(* PLC project Ackersteuerung, ForgeIEC ForgeIEC 0.1.0, author Jörg Bernau *)
(* stored: creationDateTime 2026-08-31T00:10:50 *)
(* # Ackersteuerung — Bewässerungssteuerung des SoLaWi-Ackers „Ackervielfalt"

> Automatisierte, bedarfsgerechte Bewässerung des Gemeinschaftsackers der SoLaWi Ackervielfalt
> (Kooperation mit **SALZ Automation** ). Ziel: präzises, wassersparendes Bewässern statt Handgießen.
> Ref: https://www.solawi-ackervielfalt.de/kooperation-salz-automation/
>
> Repository: https://github.com/Beerlesklopfer/Ackervielfalt — SPS-Projekt `Ackersteuerung.forge`,
> HMI-Projekt `Ackersteuerung.hearth`. **Stand 2026-09-29.**

---

## 0. Harte Randbedingungen

1. **Höchstens `Betrieb.uMaxVentile` Ventile gleichzeitig offen** (Startwert 24) — erzwungen
   durch `FB_TERMINAL_OUT` über alle Betriebsarten.
2. **Kein angewähltes Beet wird ausgelassen** — die Laufzeit zählt erst, wenn das Ventil wirklich
   offen ist; ein Beet wartet höchstens, es wird nie übersprungen.
3. **Genau eine Betriebsart** — `Betrieb.uModeActive` trägt je Betriebsart ein Bit; 0 = AUS
   (alle Ventile zu).
4. **Anwahl per HMI oder Taster** am Beet, gleichberechtigt (Dual-Namespace `Anvil.*` Hardware /
   `Bellows.*` HMI).

## 1. Anlage und Bus

Sechs Feldboxen (Amsamotion Modbus-TCP) und ein Weidmüller-UR20-Koppler, zwei Segmente an `end0`:

| Gerät | Typ | IP | Segment | Index |
|---|---|---|---|---|
| Pfirsich | ETH-MODBUS-IO8R-A | .26 | MODBUS-SUED | 0–3 |
| Stachelbeere | ETH-MODBUS-IO8R-A | .28 | MODBUS-SUED | 4–7 |
| Maulbeere | ETH-MODBUS-IO8R-A | .29 | MODBUS-SUED | 8–11 |
| Felsenbirne | ETH-MODBUS-IO8R-A | .27 | MODBUS-SUED | 12–15 |
| Maibeere | ETH-MODBUS-IO8R-A | .25 | MODBUS_NORD | 16–19 |
| Johannisbeere | ETH-MODBUS-IO8R-A | .24 | MODBUS_NORD | 20–23 |
| Schaltschrank | Weidmüller UR20-FBC-MOD-TCP (8 DI / 8 DO) | .229 | MODBUS_NORD | — |

Netz 192.168.24.x. **Alle Felder je Ventil laufen 0..23**, Index `i = z*4 + v` (Zone z in der
Reihenfolge der Tabelle, v = Taster/Ventil − 1). Die Zuordnung legt `FB_TERMINAL_OUT` fest.

## 2. Ein- und Ausgänge je Feldbox

IO8R-A (alle sechs Feldboxen): `xT_1..4` Beet-Taster · `xT_5..8` frei · `xV_1..4` Ventile ·
`xLed_5..8` Status-LEDs der Ventile 1..4 · `wAI_Voltage_1..3`, `wAI_Current_1..3`
Analogeingänge · `wAO_1..2` Analogausgänge.

## 3. Betriebsarten (`Betrieb.uModeActive`)

`PLC_PRG` ruft jeden Modus-Baustein in jedem Zyklus; sein `xEnable` entscheidet, ob er arbeitet.
Ein abgeschalteter Baustein friert ein. Dasselbe Bit setzt jeder Baustein als `bModeBit` je Ventil
in `Betrieb.astValveStatus[i].bMode`.

| Bit | Betriebsart | Baustein | Verhalten |
|---|---|---|---|
| 0 | AUS | — | nichts vorgewählt, alle Ventile und LEDs aus |
| 1 | Manuell | `fbManual` : `FB_MANUAL` | Taster oder HMI schalten das Ventil um |
| 2 | One-Shot | `fbOneShot` : `FB_SCHEDULE` | angewählte Beete laufen nach Start einmal ihre Dauer |
| 4 | wiederkehrend | `fbRecurring` : `FB_SCHEDULE` | wie One-Shot; Startzeit und Wochentage noch nicht ausgewertet (§10) |
| 8 | Auto | `fbAuto` : `FB_WEEKLY_TIMER` | Platzhalter, Bedarf nach Kc/ET0 zurückgestellt; öffnet kein Ventil |

### Lauf in One-Shot und wiederkehrend (`FB_SCHEDULE`)

- **Anwahl:** je Beet ein `JK_FF`; Feldtaster `Anvil.<Zone>.xT_v` und HMI-Puls
  `Schrittkette.axSelToggle[i]` schalten gleichberechtigt um. Q ist `Betrieb.aValveJobs[i].xSelected`.
  Nicht persistent.
- **Befehle** (je eine steigende Flanke): `Schrittkette.xStart`, `xStop`, `xPause`, `xAcknowledge`.
- **Zustand** `Schrittkette.uRunState`: 0 Idle · 1 Running · 2 Paused · 3 Done.
- **Timer:** je Beet ein `TONR` (pausierbar). Er zählt nur, solange Running und das Ventil wirklich
  offen ist; Pause und Warten auf Freigabe halten ihn an.
- **Restzeit:** `Betrieb.astValveStatus[i].remainingLiquidation` = PT − ET, nicht persistent; die HMI liest sie dort direkt.

## 4. Ausgabe und Anzeige (`FB_TERMINAL_OUT`)

`FB_TERMINAL_OUT` ist der eine Setter: Vorwahl der aktiven Betriebsart, Arbitrierung, 48 Klemmen.

- Laufende Freigaben **halten**, solange vorgewählt; neue nur bei freiem Platz, in
  Index-Reihenfolge, ohne Verdrängung.
- Fällt ein offenes Ventil, ist die Vorwahl **verbraucht** (das Bit der Betriebsart fällt).
- Ventile `xV_1..4` folgen allein der Freigabe (`astValveStatus[i].isOpen`).
- LEDs `xLed_5..8`: Dauerlicht = offen; vorgewählt und wartend = Blinken im Takt
  `Betrieb.rBlinkHz` (Startwert 0.1 Hz, begrenzt auf 0.01..10 Hz).

## 5. Persistente Einstellungen

Persistent heißt: der Wert übersteht Neustart und Programm-Download. Alle sind von der HMI
schreibbar.

| Variable | Label | Startwert | Bedeutung |
|---|---|---|---|
| `Betrieb.uModeActive` | Aktive Betriebsart | 0 | Bit der Betriebsart (§3) |
| `Betrieb.uMaxVentile` | Max. offene Ventile | 24 | Höchstzahl gleichzeitig offener Ventile |
| `Betrieb.rBlinkHz` | Blinkfrequenz wartende Ventile [Hz] | 0.1 | Blinktakt wartender Ventile |
| `Betrieb.aValveJobs` | Ventil-Jobs | Dauer 1 min | je Beet `ST_BedCfg`: Anwahl, Startzeit, Dauer |
| `Betrieb.bWeekMask` | Wochentage wiederkehrend | 0 | Bit 0 = Montag … Bit 6 = Sonntag |

**Achtung:** Gespeichert wird je Variable mit einer Typkennung. Ändert sich der Typ (ein Feld mehr
in `ST_BedCfg`, andere Feldgrenzen), verwirft der nächste Download die gespeicherten Werte dieser
Variable einmal.

## 6. HMI-Gruppen

- `Betrieb`: Einstellungen (§5) und `astValveStatus[0..23]` (`ST_ValveStatus`: bMode,
  isPreselected, isOpen, liquidationPeriod, remainingLiquidation).
- `Schrittkette`: `axSelToggle[0..23]`, die vier Befehle, `uRunState`.
- `Diag`: Geräteüberwachung (§7).
- `HmiCmd`: leer.

## 7. Geräteüberwachung

`BusMonitor` (taskDiag) liest je Gerät `Anvil.<Gerät>.Status.xOnline`, `FB_BUS_MONITOR` führt je
Gerät einen `FB_DEVICE_MONITOR` (0 Unbekannt → 1 Online → 2 Gestört → 3 Offline, entprellt) und
schreibt nach `Bellows.Diag`: `auDevState[0..6]`, `asDevStatus`, `sSummary`, `xAllOk`,
`iFaultCount`. Index 0 Pfirsich … 5 Johannisbeere, 6 Schaltschrank — handgepflegt.

## 8. Tasks

| Task | Takt | Priorität | Programm |
|---|---|---|---|
| task0 | 20 ms | 0 | `PLC_PRG` |
| taskDiag | 200 ms | 10 | `BusMonitor` |

## 9. Bausteine und Typen

Programme: `PLC_PRG`, `BusMonitor`. Funktionsbausteine: `FB_MANUAL`, `FB_SCHEDULE`,
`FB_TERMINAL_OUT`, `FB_BLINK`, `FB_WEEKLY_TIMER`, `FB_DEVICE_MONITOR`, `FB_BUS_MONITOR`.
Funktion: `FC_GetKcValue`. Aus der Standardbibliothek u. a. `JK_FF`, `TONR`, `R_TRIG`, `TON`.
Gruppen: sieben Geräte (Pfirsich … Schaltschrank) und die HMI-Gruppen `Betrieb`, `Schrittkette`,
`Diag`, `HmiCmd`.
Typen: `ST_BedCfg` (xSelected, uStartHour, uStartMin, tDuration), `ST_ValveStatus`,
`ST_KcCurve`.

## 10. Offene Punkte (2026-09-29)

- **Wochenschaltuhr:** Betriebsart wiederkehrend wertet `uStartHour`, `uStartMin` und
  `bWeekMask` noch nicht aus — sie läuft wie One-Shot auf Start. Die Dialoge zeigen bis dahin nur
  Anwahl und Dauer.
- `HmiCmd` ist leer.
- Schaltschrank: Ein- und Ausgänge ungenutzt; die Bindungen stehen in der alten Steckplatz-Zählung
  (Stand 2026-09-11, nicht neu geprüft).
- Analogausgänge `wAO_1..2`: die Bindung nennt Register 0/1, die Gerätebeschreibung 6/7
  (Stand 2026-09-11, nicht neu geprüft).
- Betriebsart Auto (Kc/ET0) wartet auf Wetter- und Bodensensorik. *)

TYPE ST_KcCurve : STRUCT
  days_initial : INT;
  days_dev : INT;
  days_mid : INT;
  days_late : INT;
  kc_initial : REAL;
  kc_mid : REAL;
  kc_end : REAL;
END_STRUCT;
END_TYPE

(* Ein Beet (ein Ventil) fuer One-Shot und wiederkehrend: Anwahl, Startzeit in Ortszeit und Bewaesserungsdauer (Vorgabe 1 min). Element der persistenten Job-Liste Betrieb.aValveJobs[0..23], Index z*4+v. xSelected schreibt die SPS (FB_SCHEDULE), Startzeit und Dauer die HMI. Die laufende Restzeit steht NICHT hier, sondern im nicht persistenten Betrieb.astValveStatus[i].remainingLiquidation — sie aendert sich jeden Zyklus, und in einem persistenten Satz schrieb sie im Lauf alle 5 s die Persistenzdatei (29.09.2026). *)
TYPE ST_BedCfg : STRUCT
  xSelected : BOOL := FALSE;  (* Wird dieses Beet bei der bewässerung berücksichtigt? *)
  uStartHour : BYTE;  (* Startzeit Stunde (Ortszeit) *)
  uStartMin : BYTE;  (* Startzeit Minute *)
  tDuration : TIME := T#1m;  (* Bewaesserungsdauer dieses Ventils, Vorgabe 1 min *)
END_STRUCT;
END_TYPE

(* Status je Ventil (Betrieb.astValveStatus, Index z*4+v). bMode: je Betriebsart ein Bit (1 Manuell, 2 One-Shot, 4 wiederkehrend, 8 Auto), von jedem Modus-Baustein in seiner Schleife gesetzt. isPreselected: vorgewaehlt in der AKTIVEN Betriebsart, (bMode AND GVL.Betrieb.uModeActive) <> 0 — schreibt FB_TERMINAL_OUT. isOpen: wirklich offen = Freigabe der Arbitrierung in FB_TERMINAL_OUT (nie mehr als uMaxVentile, laufende halten, nachruecken in Index-Reihenfolge); haelt ueber die Zyklen. liquidationPeriod: eingestellte Laufdauer, vom Modus (Manuell T#0s = unbegrenzt). remainingLiquidation: Restlauf = liquidationPeriod − ET des Modus-Timers, vom Modus berechnet. *)
TYPE ST_ValveStatus : STRUCT
  bMode : BYTE := 0;
  isPreselected : BOOL := FALSE;
  isOpen : BOOL := FALSE;
  liquidationPeriod : TIME := T#0s;
  remainingLiquidation : TIME := T#0s;
END_STRUCT;
END_TYPE

(* HMI-Gruppe Betrieb: Betriebsartwahl xManuell, xOneShot, xWiederkehrend, xAuto (genau eine gesetzt, sonst Aus), die bestaetigte Betriebsart uModeActive (0 Aus, 1 Manuell, 2 One-Shot, 3 wiederkehrend, 4 Auto) und die Einstellwerte uMaxVentile und rBlinkHz. Wahl und Einstellwerte sind persistent. *)
PROGRAM Betrieb
  VAR_GLOBAL
    uModeActive AT %MB0 : USINT := 0;  (* Aktive Betriebsart, je Betriebsart ein Bit: 0 = AUS, 1 = Manuell, 2 = One-Shot, 4 = wiederkehrend, 8 = Auto. Die EINE Quelle: PLC_PRG gibt damit die Modus-Bausteine frei (xEnable) und reicht dasselbe Bit als bModeBit weiter; FB_TERMINAL_OUT liest damit die Vorwahl aus astValveStatus[i].bMode. Von der HMI gesetzt, persistent. *)
    uMaxVentile AT %MB2 : USINT := 24;  (* Hoechstzahl gleichzeitig offener Ventile (Wasserdruck, Pumpenleistung). FB_TERMINAL_OUT begrenzt auf diese Zahl; weitere Anforderungen warten in Index-Reihenfolge und ruecken nach, sobald ein Platz frei wird. Startwert 24. Von der HMI gesetzt, persistent. *)
    rBlinkHz AT %MD7 : REAL := 0.1;  (* Blinkfrequenz der Status-LEDs wartender Ventile in den Betriebsarten Manuell, One-Shot und wiederkehrend, in Hz: angefordert, aber vom Arbiter noch nicht freigegeben. PLC_PRG begrenzt auf 0.01..10 Hz, ein Wert unter 0.01 gilt als 0.1. Startwert 0.1 Hz = 5 s an / 5 s aus. Von der HMI gesetzt, persistent. *)
  END_VAR

            
          
END_PROGRAM

(* # FB_BLINK — Blink-/Flash-Generator (Programm-Anzeige) Asymmetrisches Blinksignal aus zwei TON: kurzer Flash (`tBlFlash`) + längere Pause (`tBlPause`); `xBlQ` ist Phasen-Bit + Ausgang. `xBlEnable=FALSE` hält `xBlQ` dauerhaft FALSE (Handbetrieb blinkt nicht). In PLC_PRG mit `T#1S`/`T#29S` ( **Periode 30 s** ) für die Programm-Anzeige `xV_6..8` parametriert. Review-Hinweis: bei Enable startet die Pause zuerst (erster Flash nach `tBlPause`); `PT=0` ungeguardet. *)
FUNCTION_BLOCK FB_BLINK
  VAR
    tonBlOn : TON;  (* Timer für Flash-Dauer (tBlFlash) *)
    tonBlOff : TON;  (* Timer für Pausen-Dauer (tBlPause) *)
    xWasEnabled : BOOL;  (* Flankenspeicher xBlEnable: bei steigender Flanke startet die Anzeige mit einem Flash (sofortige Rueckmeldung) *)
  END_VAR
  VAR_INPUT
    xBlEnable : BOOL;  (* Blinken aktiv; FALSE = xBlQ dauerhaft FALSE (z. B. Handbetrieb) *)
    tBlFlash : TIME := T#1S;  (* Kurzer Flash (Ein-Dauer); relais-schonend: 1 s Flash bei 10 s Periode (1 s ein / 9 s aus) *)
    tBlPause : TIME := T#9S;  (* Laengere Pause (Aus-Dauer); relais-schonend: 9 s Pause bei 10 s Periode (1 s ein / 9 s aus) *)
  END_VAR
  VAR_OUTPUT
    xBlQ : BOOL;  (* Blink-Ausgang: kurzer Flash, längere Pause; FALSE bei NOT xBlEnable *)
  END_VAR

            (* Disable: Ausgang sofort aus, Flankenspeicher zuruecksetzen. *)
IF NOT xBlEnable THEN
    xBlQ := FALSE;
    xWasEnabled := FALSE;
ELSIF NOT xWasEnabled THEN
    (* Steigende Flanke von Enable: mit einem Flash STARTEN -> sofortige
       Rueckmeldung, kein Warten auf die erste Pause. Relais-schonend 1s/9s. *)
    xBlQ := TRUE;
    xWasEnabled := TRUE;
END_IF;

(* Zwei TON bilden den asymmetrischen Oszillator:
     - waehrend Flash (xBlQ=TRUE)  laeuft tonBlOn  (PT=tBlFlash)
     - waehrend Pause (xBlQ=FALSE) laeuft tonBlOff (PT=tBlPause) *)
tonBlOn (IN := xBlEnable AND xBlQ,     PT := tBlFlash);
tonBlOff(IN := xBlEnable AND NOT xBlQ, PT := tBlPause);

IF xBlEnable THEN
    IF xBlQ AND tonBlOn.Q THEN
        xBlQ := FALSE;          (* Flash zu Ende -> Pause beginnt *)
    ELSIF (NOT xBlQ) AND tonBlOff.Q THEN
        xBlQ := TRUE;           (* Pause zu Ende -> Flash beginnt *)
    END_IF;
END_IF;
          
END_FUNCTION_BLOCK

(* Feldbox Felsenbirne (Amsamotion ETH-MODBUS-IO8R-A, 192.168.24.27, Segment MODBUS-SUED), Ventile 13-16 der Job-Liste. xT_1..4 Beet-Taster, xT_5..8 frei; xV_1..4 Ventile (= Arbiter-Freigabe); xV_5..8 Status-LEDs der Ventile 1..4; wAI_Voltage_1..3 und wAI_Current_1..3 Analogeingaenge; wAO_1..2 Analogausgaenge. Anvil.* ist die Hardware-Sicht, Bellows.* die HMI-Sicht derselben Variablen. *)
PROGRAM Felsenbirne
  VAR_GLOBAL
    xT_1 AT %IX5.0 : BOOL;  (* Digital input channel 1 (24V DC, opto-isolated) *)
    xT_2 AT %IX5.1 : BOOL;  (* Digital input channel 2 (24V DC, opto-isolated) *)
    xT_3 AT %IX5.2 : BOOL;  (* Digital input channel 3 (24V DC, opto-isolated) *)
    xT_4 AT %IX5.3 : BOOL;  (* Digital input channel 4 (24V DC, opto-isolated) *)
    xT_5 AT %IX5.4 : BOOL;  (* Digital input channel 5 (24V DC, opto-isolated) *)
    xT_6 AT %IX5.5 : BOOL;  (* Digital input channel 6 (24V DC, opto-isolated) *)
    xT_7 AT %IX5.6 : BOOL;  (* Digital input channel 7 (24V DC, opto-isolated) *)
    xT_8 AT %IX5.7 : BOOL;  (* Digital input channel 8 (24V DC, opto-isolated) *)
    xV_1 AT %QX5.0 : BOOL;  (* Relay output channel 1 (max 2A) *)
    xV_2 AT %QX5.1 : BOOL;  (* Relay output channel 2 (max 2A) *)
    xV_3 AT %QX5.2 : BOOL;  (* Relay output channel 3 (max 2A) *)
    xV_4 AT %QX5.3 : BOOL;  (* Relay output channel 4 (max 2A) *)
    xLed_5 AT %QX5.4 : BOOL;  (* Relay output channel 5 (max 2A) *)
    xLed_6 AT %QX5.5 : BOOL;  (* Relay output channel 6 (max 2A) *)
    xLed_7 AT %QX5.6 : BOOL;  (* Relay output channel 7 (max 2A) *)
    xLed_8 AT %QX5.7 : BOOL;  (* Relay output channel 8 (max 2A) *)
    wAO_1 AT %QW8 : UINT;  (* Analog output channel 1 (0-10V / 0-20mA, 12-bit) *)
    wAO_2 AT %QW9 : UINT;  (* Analog output channel 2 (0-10V / 0-20mA, 12-bit) *)
    wAI_Voltage_1 AT %IW24 : UINT;  (* Analog input channel 1 (0-10V, 12-bit) *)
    wAI_Voltage_2 AT %IW25 : UINT;  (* Analog input channel 2 (0-10V, 12-bit) *)
    wAI_Voltage_3 AT %IW26 : UINT;  (* Analog input channel 3 (0-10V, 12-bit) *)
    wAI_Current_1 AT %IW27 : UINT;  (* Analog input channel 4 (0-20mA, 12-bit) *)
    wAI_Current_2 AT %IW28 : UINT;  (* Analog input channel 5 (0-20mA, 12-bit) *)
    wAI_Current_3 AT %IW29 : UINT;  (* Analog input channel 6 (0-20mA, 12-bit) *)
  END_VAR

            
          
END_PROGRAM

(* Feldbox Johannisbeere (Amsamotion ETH-MODBUS-IO8R-A, 192.168.24.24, Segment MODBUS_NORD), Ventile 21-24 der Job-Liste. xT_1..4 Beet-Taster, xT_5..8 frei; xV_1..4 Ventile (= Arbiter-Freigabe); xV_5..8 Status-LEDs der Ventile 1..4; wAI_Voltage_1..3 und wAI_Current_1..3 Analogeingaenge; wAO_1..2 Analogausgaenge. Anvil.* ist die Hardware-Sicht, Bellows.* die HMI-Sicht derselben Variablen. *)
PROGRAM Johannisbeere
  VAR_GLOBAL
    xT_1 AT %IX4.0 : BOOL;  (* Digital input channel 1 (24V DC, opto-isolated) *)
    xT_2 AT %IX4.1 : BOOL;  (* Digital input channel 2 (24V DC, opto-isolated) *)
    xT_3 AT %IX4.2 : BOOL;  (* Digital input channel 3 (24V DC, opto-isolated) *)
    xT_4 AT %IX4.3 : BOOL;  (* Digital input channel 4 (24V DC, opto-isolated) *)
    xT_5 AT %IX4.4 : BOOL;  (* Digital input channel 5 (24V DC, opto-isolated) *)
    xT_6 AT %IX4.5 : BOOL;  (* Digital input channel 6 (24V DC, opto-isolated) *)
    xT_7 AT %IX4.6 : BOOL;  (* Digital input channel 7 (24V DC, opto-isolated) *)
    xT_8 AT %IX4.7 : BOOL;  (* Digital input channel 8 (24V DC, opto-isolated) *)
    xV_1 AT %QX4.0 : BOOL;  (* Relay output channel 1 (max 2A) *)
    xV_2 AT %QX4.1 : BOOL;  (* Relay output channel 2 (max 2A) *)
    xV_3 AT %QX4.2 : BOOL;  (* Relay output channel 3 (max 2A) *)
    xV_4 AT %QX4.3 : BOOL;  (* Relay output channel 4 (max 2A) *)
    xLed_5 AT %QX4.4 : BOOL;  (* Relay output channel 5 (max 2A) *)
    xLed_6 AT %QX4.5 : BOOL;  (* Relay output channel 6 (max 2A) *)
    xLed_7 AT %QX4.6 : BOOL;  (* Relay output channel 7 (max 2A) *)
    xLed_8 AT %QX4.7 : BOOL;  (* Relay output channel 8 (max 2A) *)
    wAI_Voltage_1 AT %IW18 : UINT;  (* Analog input channel 1 (0-10V, 12-bit) *)
    wAI_Voltage_2 AT %IW19 : UINT;  (* Analog input channel 2 (0-10V, 12-bit) *)
    wAI_Voltage_3 AT %IW20 : UINT;  (* Analog input channel 3 (0-10V, 12-bit) *)
    wAI_Current_1 AT %IW21 : UINT;  (* Analog input channel 4 (0-20mA, 12-bit) *)
    wAI_Current_2 AT %IW22 : UINT;  (* Analog input channel 5 (0-20mA, 12-bit) *)
    wAI_Current_3 AT %IW23 : UINT;  (* Analog input channel 6 (0-20mA, 12-bit) *)
    wAO_1 AT %QW6 : UINT;  (* Analog output channel 1 (0-10V / 0-20mA, 12-bit) *)
    wAO_2 AT %QW7 : UINT;  (* Analog output channel 2 (0-10V / 0-20mA, 12-bit) *)
  END_VAR

            
          
END_PROGRAM

(* Feldbox Maibeere (Amsamotion ETH-MODBUS-IO8R-A, 192.168.24.25, Segment MODBUS_NORD), Ventile 17-20 der Job-Liste. xT_1..4 Beet-Taster, xT_5..8 frei; xV_1..4 Ventile (= Arbiter-Freigabe); xV_5..8 Status-LEDs der Ventile 1..4; wAI_Voltage_1..3 und wAI_Current_1..3 Analogeingaenge; wAO_1..2 Analogausgaenge. Anvil.* ist die Hardware-Sicht, Bellows.* die HMI-Sicht derselben Variablen. *)
PROGRAM Maibeere
  VAR_GLOBAL
    xT_1 AT %IX3.0 : BOOL;  (* Digital input channel 1 (24V DC, opto-isolated) *)
    xT_2 AT %IX3.1 : BOOL;  (* Digital input channel 2 (24V DC, opto-isolated) *)
    xT_3 AT %IX3.2 : BOOL;  (* Digital input channel 3 (24V DC, opto-isolated) *)
    xT_4 AT %IX3.3 : BOOL;  (* Digital input channel 4 (24V DC, opto-isolated) *)
    xT_5 AT %IX3.4 : BOOL;  (* Digital input channel 5 (24V DC, opto-isolated) *)
    xT_6 AT %IX3.5 : BOOL;  (* Digital input channel 6 (24V DC, opto-isolated) *)
    xT_7 AT %IX3.6 : BOOL;  (* Digital input channel 7 (24V DC, opto-isolated) *)
    xT_8 AT %IX3.7 : BOOL;  (* Digital input channel 8 (24V DC, opto-isolated) *)
    xV_1 AT %QX3.0 : BOOL;  (* Relay output channel 1 (max 2A) *)
    xV_2 AT %QX3.1 : BOOL;  (* Relay output channel 2 (max 2A) *)
    xV_3 AT %QX3.2 : BOOL;  (* Relay output channel 3 (max 2A) *)
    xV_4 AT %QX3.3 : BOOL;  (* Relay output channel 4 (max 2A) *)
    xLed_5 AT %QX3.4 : BOOL;  (* Relay output channel 5 (max 2A) *)
    xLed_6 AT %QX3.5 : BOOL;  (* Relay output channel 6 (max 2A) *)
    xLed_7 AT %QX3.6 : BOOL;  (* Relay output channel 7 (max 2A) *)
    xLed_8 AT %QX3.7 : BOOL;  (* Relay output channel 8 (max 2A) *)
    wAI_Voltage_1 AT %IW30 : UINT;  (* Analog input channel 1 (0-10V, 12-bit) *)
    wAI_Voltage_2 AT %IW31 : UINT;  (* Analog input channel 2 (0-10V, 12-bit) *)
    wAI_Voltage_3 AT %IW32 : UINT;  (* Analog input channel 3 (0-10V, 12-bit) *)
    wAI_Current_1 AT %IW33 : UINT;  (* Analog input channel 4 (0-20mA, 12-bit) *)
    wAI_Current_2 AT %IW34 : UINT;  (* Analog input channel 5 (0-20mA, 12-bit) *)
    wAI_Current_3 AT %IW35 : UINT;  (* Analog input channel 6 (0-20mA, 12-bit) *)
    wAO_1 AT %QW10 : UINT;  (* Analog output channel 1 (0-10V / 0-20mA, 12-bit) *)
    wAO_2 AT %QW11 : UINT;  (* Analog output channel 2 (0-10V / 0-20mA, 12-bit) *)
  END_VAR

            
          
END_PROGRAM

(* Feldbox Maulbeere (Amsamotion ETH-MODBUS-IO8R-A, 192.168.24.29, Segment MODBUS-SUED), Ventile 9-12 der Job-Liste. xT_1..4 Beet-Taster, xT_5..8 frei; xV_1..4 Ventile (= Arbiter-Freigabe); xV_5..8 Status-LEDs der Ventile 1..4; wAI_Voltage_1..3 und wAI_Current_1..3 Analogeingaenge; wAO_1..2 Analogausgaenge. Anvil.* ist die Hardware-Sicht, Bellows.* die HMI-Sicht derselben Variablen. *)
PROGRAM Maulbeere
  VAR_GLOBAL
    xT_1 AT %IX2.0 : BOOL;  (* Digital input channel 1 (24V DC, opto-isolated) *)
    xT_2 AT %IX2.1 : BOOL;  (* Digital input channel 2 (24V DC, opto-isolated) *)
    xT_3 AT %IX2.2 : BOOL;  (* Digital input channel 3 (24V DC, opto-isolated) *)
    xT_4 AT %IX2.3 : BOOL;  (* Digital input channel 4 (24V DC, opto-isolated) *)
    xT_5 AT %IX2.4 : BOOL;  (* Digital input channel 5 (24V DC, opto-isolated) *)
    xT_6 AT %IX2.5 : BOOL;  (* Digital input channel 6 (24V DC, opto-isolated) *)
    xT_7 AT %IX2.6 : BOOL;  (* Digital input channel 7 (24V DC, opto-isolated) *)
    xT_8 AT %IX2.7 : BOOL;  (* Digital input channel 8 (24V DC, opto-isolated) *)
    xV_1 AT %QX2.0 : BOOL;  (* Relay output channel 1 (max 2A) *)
    xV_2 AT %QX2.1 : BOOL;  (* Relay output channel 2 (max 2A) *)
    xV_3 AT %QX2.2 : BOOL;  (* Relay output channel 3 (max 2A) *)
    xV_4 AT %QX2.3 : BOOL;  (* Relay output channel 4 (max 2A) *)
    xLed_5 AT %QX2.4 : BOOL;  (* Relay output channel 5 (max 2A) *)
    xLed_6 AT %QX2.5 : BOOL;  (* Relay output channel 6 (max 2A) *)
    xLed_7 AT %QX2.6 : BOOL;  (* Relay output channel 7 (max 2A) *)
    xLed_8 AT %QX2.7 : BOOL;  (* Relay output channel 8 (max 2A) *)
    wAI_Voltage_1 AT %IW12 : UINT;  (* Analog input channel 1 (0-10V, 12-bit) *)
    wAI_Voltage_2 AT %IW13 : UINT;  (* Analog input channel 2 (0-10V, 12-bit) *)
    wAI_Voltage_3 AT %IW14 : UINT;  (* Analog input channel 3 (0-10V, 12-bit) *)
    wAI_Current_1 AT %IW15 : UINT;  (* Analog input channel 4 (0-20mA, 12-bit) *)
    wAI_Current_2 AT %IW16 : UINT;  (* Analog input channel 5 (0-20mA, 12-bit) *)
    wAI_Current_3 AT %IW17 : UINT;  (* Analog input channel 6 (0-20mA, 12-bit) *)
    wAO_1 AT %QW4 : UINT;  (* Analog output channel 1 (0-10V / 0-20mA, 12-bit) *)
    wAO_2 AT %QW5 : UINT;  (* Analog output channel 2 (0-10V / 0-20mA, 12-bit) *)
  END_VAR

            
          
END_PROGRAM

(* Feldbox Pfirsich (Amsamotion ETH-MODBUS-IO8R-A, 192.168.24.26, Segment MODBUS-SUED), Ventile 1-4 der Job-Liste. xT_1..4 Beet-Taster, xT_5..8 frei; xV_1..4 Ventile (= Arbiter-Freigabe); xV_5..8 Status-LEDs der Ventile 1..4; wAI_Voltage_1..3 und wAI_Current_1..3 Analogeingaenge; wAO_1..2 Analogausgaenge. Anvil.* ist die Hardware-Sicht, Bellows.* die HMI-Sicht derselben Variablen. *)
PROGRAM Pfirsich
  VAR_GLOBAL
    xT_1 AT %IX0.0 : BOOL;  (* Digital input channel 1 (24V DC, opto-isolated) *)
    xT_2 AT %IX0.1 : BOOL;  (* Digital input channel 2 (24V DC, opto-isolated) *)
    xT_3 AT %IX0.2 : BOOL;  (* Digital input channel 3 (24V DC, opto-isolated) *)
    xT_4 AT %IX0.3 : BOOL;  (* Digital input channel 4 (24V DC, opto-isolated) *)
    xT_5 AT %IX0.4 : BOOL;  (* Digital input channel 5 (24V DC, opto-isolated) *)
    xT_6 AT %IX0.5 : BOOL;  (* Digital input channel 6 (24V DC, opto-isolated) *)
    xT_7 AT %IX0.6 : BOOL;  (* Digital input channel 7 (24V DC, opto-isolated) *)
    xT_8 AT %IX0.7 : BOOL;  (* Digital input channel 8 (24V DC, opto-isolated) *)
    xV_1 AT %QX0.0 : BOOL;  (* Relay output channel 1 (max 2A) *)
    xV_2 AT %QX0.1 : BOOL;  (* Relay output channel 2 (max 2A) *)
    xV_3 AT %QX0.2 : BOOL;  (* Relay output channel 3 (max 2A) *)
    xV_4 AT %QX0.3 : BOOL;  (* Relay output channel 4 (max 2A) *)
    xLed_5 AT %QX0.4 : BOOL;  (* Relay output channel 5 (max 2A) *)
    xLed_6 AT %QX0.5 : BOOL;  (* Relay output channel 6 (max 2A) *)
    xLed_7 AT %QX0.6 : BOOL;  (* Relay output channel 7 (max 2A) *)
    xLed_8 AT %QX0.7 : BOOL;  (* Relay output channel 8 (max 2A) *)
    wAI_Voltage_1 AT %IW0 : UINT;  (* Analog input channel 1 (0-10V, 12-bit) *)
    wAI_Voltage_2 AT %IW1 : UINT;  (* Analog input channel 2 (0-10V, 12-bit) *)
    wAI_Voltage_3 AT %IW2 : UINT;  (* Analog input channel 3 (0-10V, 12-bit) *)
    wAI_Current_1 AT %IW3 : UINT;  (* Analog input channel 4 (0-20mA, 12-bit) *)
    wAI_Current_2 AT %IW4 : UINT;  (* Analog input channel 5 (0-20mA, 12-bit) *)
    wAI_Current_3 AT %IW5 : UINT;  (* Analog input channel 6 (0-20mA, 12-bit) *)
    wAO_1 AT %QW0 : UINT;  (* Analog output channel 1 (0-10V / 0-20mA, 12-bit) *)
    wAO_2 AT %QW1 : UINT;  (* Analog output channel 2 (0-10V / 0-20mA, 12-bit) *)
  END_VAR

            
          
END_PROGRAM

(* HMI-Gruppe Schrittkette: Anwahl-Puls je Beet (axSelToggle, Index z*4+v, 0..23), die Befehle xStart, xStop, xPause und xAcknowledge (FB_SCHEDULE wertet je eine steigende Flanke aus) und der Laufzustand uRunState (0 Idle, 1 Running, 2 Paused, 3 Done). Die Restzeit je Beet steht in Betrieb.astValveStatus[i].remainingLiquidation (nicht persistent). Den Warterang (auQueue) gibt es nicht mehr. *)
PROGRAM Schrittkette
  VAR_GLOBAL
    xStart AT %MX0.5 : BOOL;  (* HMI-Startimpuls One-Shot-Schrittkette (Puls via Handshake). Steigende Flanke armt die selektierten Beete. *)
    xStop AT %MX0.6 : BOOL;  (* HMI-Stop One-Shot-Schrittkette (Puls via Handshake). Bricht den laufenden Lauf ab: alle Ventile zu, Schritte -> idle; neuer Start noetig. *)
    xPause AT %MX0.7 : BOOL;  (* HMI-Pause One-Shot-Schrittkette (Halten/Toggle via Handshake). Pause: Ventile zu + Restzeit-Timer eingefroren; erneut = fortsetzen (Ventile wieder auf). *)
    xAcknowledge AT %MX1.0 : BOOL;  (* HMI-Quittieren One-Shot-Schrittkette (Puls via Handshake). Loescht den Fertig-/Stoerungs-Status (xSeqAllDone) nach einem Lauf. *)
    axSelToggle AT %MD6 : ARRAY[0..23] OF BOOL;  (* HMI-Anwahl-Puls je Beet (momentan, schreibbar), Index z*4+v wie Betrieb.astValveStatus (0..23). Beet-Taster im Bild und Vorwahl-Haken im Dialog geben denselben Puls; FB_SCHEDULE kippt daraus Betrieb.aValveJobs[].xSelected. Ersetzt das Schreiben auf den nicht-schreibbaren Anvil-Taster xT. *)
  END_VAR

            
          
END_PROGRAM

(* Feldbox Stachelbeere (Amsamotion ETH-MODBUS-IO8R-A, 192.168.24.28, Segment MODBUS-SUED), Ventile 5-8 der Job-Liste. xT_1..4 Beet-Taster, xT_5..8 frei; xV_1..4 Ventile (= Arbiter-Freigabe); xV_5..8 Status-LEDs der Ventile 1..4; wAI_Voltage_1..3 und wAI_Current_1..3 Analogeingaenge; wAO_1..2 Analogausgaenge. Anvil.* ist die Hardware-Sicht, Bellows.* die HMI-Sicht derselben Variablen. *)
PROGRAM Stachelbeere
  VAR_GLOBAL
    xT_1 AT %IX1.0 : BOOL;  (* Digital input channel 1 (24V DC, opto-isolated) *)
    xT_2 AT %IX1.1 : BOOL;  (* Digital input channel 2 (24V DC, opto-isolated) *)
    xT_3 AT %IX1.2 : BOOL;  (* Digital input channel 3 (24V DC, opto-isolated) *)
    xT_4 AT %IX1.3 : BOOL;  (* Digital input channel 4 (24V DC, opto-isolated) *)
    xT_5 AT %IX1.4 : BOOL;  (* Digital input channel 5 (24V DC, opto-isolated) *)
    xT_6 AT %IX1.5 : BOOL;  (* Digital input channel 6 (24V DC, opto-isolated) *)
    xT_7 AT %IX1.6 : BOOL;  (* Digital input channel 7 (24V DC, opto-isolated) *)
    xT_8 AT %IX1.7 : BOOL;  (* Digital input channel 8 (24V DC, opto-isolated) *)
    xV_1 AT %QX1.0 : BOOL;  (* Relay output channel 1 (max 2A) *)
    xV_2 AT %QX1.1 : BOOL;  (* Relay output channel 2 (max 2A) *)
    xV_3 AT %QX1.2 : BOOL;  (* Relay output channel 3 (max 2A) *)
    xV_4 AT %QX1.3 : BOOL;  (* Relay output channel 4 (max 2A) *)
    xLed_5 AT %QX1.4 : BOOL;  (* Relay output channel 5 (max 2A) *)
    xLed_6 AT %QX1.5 : BOOL;  (* Relay output channel 6 (max 2A) *)
    xLed_7 AT %QX1.6 : BOOL;  (* Relay output channel 7 (max 2A) *)
    xLed_8 AT %QX1.7 : BOOL;  (* Relay output channel 8 (max 2A) *)
    wAI_Voltage_1 AT %IW6 : UINT;  (* Analog input channel 1 (0-10V, 12-bit) *)
    wAI_Voltage_2 AT %IW7 : UINT;  (* Analog input channel 2 (0-10V, 12-bit) *)
    wAI_Voltage_3 AT %IW8 : UINT;  (* Analog input channel 3 (0-10V, 12-bit) *)
    wAI_Current_1 AT %IW9 : UINT;  (* Analog input channel 4 (0-20mA, 12-bit) *)
    wAI_Current_2 AT %IW10 : UINT;  (* Analog input channel 5 (0-20mA, 12-bit) *)
    wAI_Current_3 AT %IW11 : UINT;  (* Analog input channel 6 (0-20mA, 12-bit) *)
    wAO_1 AT %QW2 : UINT;  (* Analog output channel 1 (0-10V / 0-20mA, 12-bit) *)
    wAO_2 AT %QW3 : UINT;  (* Analog output channel 2 (0-10V / 0-20mA, 12-bit) *)
  END_VAR

            
          
END_PROGRAM

FUNCTION_BLOCK FB_TERMINAL_OUT
  VAR
    fbBlink : FB_BLINK;  (* Blinktakt fuer angeforderte, aber nicht freigegebene Ventile; symmetrisch aus Betrieb.rBlinkHz. *)
    atRun : ARRAY[0..23] OF TON;  (* Je Ventil ein Laufzeit-Timer: IN = Freigabe, ET = bisheriger Lauf (currentLiquidation). Faellt die Freigabe, faellt ET. *)
    i : INT;  (* Laufindex ueber die 24 Ventile. *)
    n : DINT;  (* Zaehler der Arbitrierung (offene Ventile gegen uMaxVentile) und danach die halbe Blinkperiode in ms. *)
  END_VAR
  VAR_INPUT
    xEnable : BOOL;  (* Der einzige Anschluss. FALSE = alle 48 Klemmen AUS — kein Einfrieren: ein Ausgabe-Baustein, der stehen bleibt, liesse Ventile offen. *)
  END_VAR

            (* ============================================================================
   FB_TERMINAL_OUT  —  Der eine Setter: Arbitrierung auf der DUT, dann 48 Klemmen
   ----------------------------------------------------------------------------
   Projekt : Ackersteuerung (SoLaWi-Acker Bewaesserung)
   Autor   : Joerg Bernau / Blacksmith
   Datum   : 2026-09-22
   ----------------------------------------------------------------------------
   Der Zustand je Ventil ist Bellows.Betrieb.astValveStatus[i], Index z*4+v:
        bMode                je Betriebsart ein Bit, von den Modus-Bausteinen
        isPreselected        vorgewaehlt in der AKTIVEN Betriebsart
                             = (bMode AND GVL.Betrieb.uModeActive) <> 0
        isOpen               wirklich offen = Freigabe; haelt ueber die Zyklen
        liquidationPeriod    eingestellte Laufdauer, vom Modus (Manuell T#0s)
        remainingLiquidation Restlauf = liquidationPeriod - ET, vom Modus

   ARBITRIERUNG (ehemals FB_VALVE_ARBITER): nie mehr als uMaxVentile Ventile
   gleichzeitig offen. Laufende Freigaben HALTEN, solange vorgewaehlt; neue
   nur bei freiem Platz, in Index-Reihenfolge, keine Verdraengung. Einen
   Warterang gibt es nicht mehr (Schrittkette.auQueue entfernt 2026-09-28:
   geschrieben, von niemandem gelesen).

   DIE VORWAHL WIRD VOM LAUF VERBRAUCHT: faellt ein offenes Ventil (Flanke
   auf isOpen), loescht der Setter das Bit der aktiven Betriebsart in bMode —
   die Vorwahl faellt, das Ventil stellt sich nicht wieder an. Der Modus
   nimmt die Abwahl an (FB_MANUAL: RESET am JK_FF, wenn sein Bit fehlt).

   xEnable = FALSE (Betriebsart AUS): nichts ist vorgewaehlt, jede Freigabe
   faellt, alle 48 Klemmen AUS — kein Einfrieren.

   LED: offen = Dauerlicht, vorgewaehlt und wartend = Blink. Der Takt kommt
   aus Betrieb.rBlinkHz (0.01..10 Hz, darunter 0.1 Hz), halbe Periode in ms.

   Index z*4+v, Reihenfolge Pfirsich, Stachelbeere, Maulbeere, Felsenbirne,
   Maibeere, Johannisbeere. Seit 2026-09-28 laufen ALLE Felder je Ventil
   0..23 (astValveStatus, aValveJobs, axSelToggle).
   ============================================================================ *)

(* --- 1) Vorwahl: das Bit der aktiven Betriebsart, bei AUS nichts --- *)
FOR i := 0 TO 23 DO
    Bellows.Betrieb.astValveStatus[i].isPreselected := xEnable AND
        ((Bellows.Betrieb.astValveStatus[i].bMode AND GVL.Betrieb.uModeActive) <> 0);
END_FOR;

(* --- 2) Laufende Freigaben halten, solange vorgewaehlt und Platz ist.
       Faellt eine: die Vorwahl ist verbraucht. --- *)
n := 0;
FOR i := 0 TO 23 DO
    IF Bellows.Betrieb.astValveStatus[i].isOpen
       AND Bellows.Betrieb.astValveStatus[i].isPreselected
       AND (n < USINT_TO_DINT(GVL.Betrieb.uMaxVentile)) THEN
        n := n + 1;
    ELSE
        IF Bellows.Betrieb.astValveStatus[i].isOpen THEN
            Bellows.Betrieb.astValveStatus[i].bMode :=
                Bellows.Betrieb.astValveStatus[i].bMode AND NOT GVL.Betrieb.uModeActive;
            Bellows.Betrieb.astValveStatus[i].isPreselected := FALSE;
        END_IF;
        Bellows.Betrieb.astValveStatus[i].isOpen := FALSE;
    END_IF;
END_FOR;

(* --- 3) Nachruecken: vorgewaehlt, noch zu, Platz frei — in Index-Reihenfolge --- *)
FOR i := 0 TO 23 DO
    IF Bellows.Betrieb.astValveStatus[i].isPreselected
       AND NOT Bellows.Betrieb.astValveStatus[i].isOpen
       AND (n < USINT_TO_DINT(GVL.Betrieb.uMaxVentile)) THEN
        Bellows.Betrieb.astValveStatus[i].isOpen := TRUE;
        n := n + 1;
    END_IF;
END_FOR;

(* --- 4) Blinktakt fuer die Wartenden: halbe Periode in ms aus rBlinkHz --- *)
n := 5000;
IF GVL.Betrieb.rBlinkHz >= 0.01 THEN
    n := REAL_TO_DINT(500.0 / GVL.Betrieb.rBlinkHz);
END_IF;
IF n < 50 THEN
    n := 50;
END_IF;
fbBlink(xBlEnable := xEnable, tBlFlash := DINT_TO_TIME(n), tBlPause := DINT_TO_TIME(n));

(* --- 5) Die Ventilklemmen: offen = Freigabe --- *)
Anvil.Pfirsich.xV_1 := Bellows.Betrieb.astValveStatus[0].isOpen;
Anvil.Pfirsich.xV_2 := Bellows.Betrieb.astValveStatus[1].isOpen;
Anvil.Pfirsich.xV_3 := Bellows.Betrieb.astValveStatus[2].isOpen;
Anvil.Pfirsich.xV_4 := Bellows.Betrieb.astValveStatus[3].isOpen;

Anvil.Stachelbeere.xV_1 := Bellows.Betrieb.astValveStatus[4].isOpen;
Anvil.Stachelbeere.xV_2 := Bellows.Betrieb.astValveStatus[5].isOpen;
Anvil.Stachelbeere.xV_3 := Bellows.Betrieb.astValveStatus[6].isOpen;
Anvil.Stachelbeere.xV_4 := Bellows.Betrieb.astValveStatus[7].isOpen;

Anvil.Maulbeere.xV_1 := Bellows.Betrieb.astValveStatus[8].isOpen;
Anvil.Maulbeere.xV_2 := Bellows.Betrieb.astValveStatus[9].isOpen;
Anvil.Maulbeere.xV_3 := Bellows.Betrieb.astValveStatus[10].isOpen;
Anvil.Maulbeere.xV_4 := Bellows.Betrieb.astValveStatus[11].isOpen;

Anvil.Felsenbirne.xV_1 := Bellows.Betrieb.astValveStatus[12].isOpen;
Anvil.Felsenbirne.xV_2 := Bellows.Betrieb.astValveStatus[13].isOpen;
Anvil.Felsenbirne.xV_3 := Bellows.Betrieb.astValveStatus[14].isOpen;
Anvil.Felsenbirne.xV_4 := Bellows.Betrieb.astValveStatus[15].isOpen;

Anvil.Maibeere.xV_1 := Bellows.Betrieb.astValveStatus[16].isOpen;
Anvil.Maibeere.xV_2 := Bellows.Betrieb.astValveStatus[17].isOpen;
Anvil.Maibeere.xV_3 := Bellows.Betrieb.astValveStatus[18].isOpen;
Anvil.Maibeere.xV_4 := Bellows.Betrieb.astValveStatus[19].isOpen;

Anvil.Johannisbeere.xV_1 := Bellows.Betrieb.astValveStatus[20].isOpen;
Anvil.Johannisbeere.xV_2 := Bellows.Betrieb.astValveStatus[21].isOpen;
Anvil.Johannisbeere.xV_3 := Bellows.Betrieb.astValveStatus[22].isOpen;
Anvil.Johannisbeere.xV_4 := Bellows.Betrieb.astValveStatus[23].isOpen;

(* --- 6) Die LED-Klemmen: offen = an, vorgewaehlt und wartend = Blink --- *)
Anvil.Pfirsich.xLed_5 := Bellows.Betrieb.astValveStatus[0].isOpen OR (Bellows.Betrieb.astValveStatus[0].isPreselected AND fbBlink.xBlQ);
Anvil.Pfirsich.xLed_6 := Bellows.Betrieb.astValveStatus[1].isOpen OR (Bellows.Betrieb.astValveStatus[1].isPreselected AND fbBlink.xBlQ);
Anvil.Pfirsich.xLed_7 := Bellows.Betrieb.astValveStatus[2].isOpen OR (Bellows.Betrieb.astValveStatus[2].isPreselected AND fbBlink.xBlQ);
Anvil.Pfirsich.xLed_8 := Bellows.Betrieb.astValveStatus[3].isOpen OR (Bellows.Betrieb.astValveStatus[3].isPreselected AND fbBlink.xBlQ);

Anvil.Stachelbeere.xLed_5 := Bellows.Betrieb.astValveStatus[4].isOpen OR (Bellows.Betrieb.astValveStatus[4].isPreselected AND fbBlink.xBlQ);
Anvil.Stachelbeere.xLed_6 := Bellows.Betrieb.astValveStatus[5].isOpen OR (Bellows.Betrieb.astValveStatus[5].isPreselected AND fbBlink.xBlQ);
Anvil.Stachelbeere.xLed_7 := Bellows.Betrieb.astValveStatus[6].isOpen OR (Bellows.Betrieb.astValveStatus[6].isPreselected AND fbBlink.xBlQ);
Anvil.Stachelbeere.xLed_8 := Bellows.Betrieb.astValveStatus[7].isOpen OR (Bellows.Betrieb.astValveStatus[7].isPreselected AND fbBlink.xBlQ);

Anvil.Maulbeere.xLed_5 := Bellows.Betrieb.astValveStatus[8].isOpen OR (Bellows.Betrieb.astValveStatus[8].isPreselected AND fbBlink.xBlQ);
Anvil.Maulbeere.xLed_6 := Bellows.Betrieb.astValveStatus[9].isOpen OR (Bellows.Betrieb.astValveStatus[9].isPreselected AND fbBlink.xBlQ);
Anvil.Maulbeere.xLed_7 := Bellows.Betrieb.astValveStatus[10].isOpen OR (Bellows.Betrieb.astValveStatus[10].isPreselected AND fbBlink.xBlQ);
Anvil.Maulbeere.xLed_8 := Bellows.Betrieb.astValveStatus[11].isOpen OR (Bellows.Betrieb.astValveStatus[11].isPreselected AND fbBlink.xBlQ);

Anvil.Felsenbirne.xLed_5 := Bellows.Betrieb.astValveStatus[12].isOpen OR (Bellows.Betrieb.astValveStatus[12].isPreselected AND fbBlink.xBlQ);
Anvil.Felsenbirne.xLed_6 := Bellows.Betrieb.astValveStatus[13].isOpen OR (Bellows.Betrieb.astValveStatus[13].isPreselected AND fbBlink.xBlQ);
Anvil.Felsenbirne.xLed_7 := Bellows.Betrieb.astValveStatus[14].isOpen OR (Bellows.Betrieb.astValveStatus[14].isPreselected AND fbBlink.xBlQ);
Anvil.Felsenbirne.xLed_8 := Bellows.Betrieb.astValveStatus[15].isOpen OR (Bellows.Betrieb.astValveStatus[15].isPreselected AND fbBlink.xBlQ);

Anvil.Maibeere.xLed_5 := Bellows.Betrieb.astValveStatus[16].isOpen OR (Bellows.Betrieb.astValveStatus[16].isPreselected AND fbBlink.xBlQ);
Anvil.Maibeere.xLed_6 := Bellows.Betrieb.astValveStatus[17].isOpen OR (Bellows.Betrieb.astValveStatus[17].isPreselected AND fbBlink.xBlQ);
Anvil.Maibeere.xLed_7 := Bellows.Betrieb.astValveStatus[18].isOpen OR (Bellows.Betrieb.astValveStatus[18].isPreselected AND fbBlink.xBlQ);
Anvil.Maibeere.xLed_8 := Bellows.Betrieb.astValveStatus[19].isOpen OR (Bellows.Betrieb.astValveStatus[19].isPreselected AND fbBlink.xBlQ);

Anvil.Johannisbeere.xLed_5 := Bellows.Betrieb.astValveStatus[20].isOpen OR (Bellows.Betrieb.astValveStatus[20].isPreselected AND fbBlink.xBlQ);
Anvil.Johannisbeere.xLed_6 := Bellows.Betrieb.astValveStatus[21].isOpen OR (Bellows.Betrieb.astValveStatus[21].isPreselected AND fbBlink.xBlQ);
Anvil.Johannisbeere.xLed_7 := Bellows.Betrieb.astValveStatus[22].isOpen OR (Bellows.Betrieb.astValveStatus[22].isPreselected AND fbBlink.xBlQ);
Anvil.Johannisbeere.xLed_8 := Bellows.Betrieb.astValveStatus[23].isOpen OR (Bellows.Betrieb.astValveStatus[23].isPreselected AND fbBlink.xBlQ);

          
END_FUNCTION_BLOCK

(* # FB_MANUAL — Handbetrieb, Betriebsart 1 `FB_MANUAL` bildet den Handbetrieb fuer 24 Ventile ab. Der Baustein wird zyklisch von `PLC_PRG` aufgerufen und liefert zwei Muster zurueck: - `axValve[0..23]`: angewaehlte Ventile im Handbetrieb - `axLed[0..23]`: zugehoeriges Lampenmuster, aktuell identisch zu `axValve` Die Reihenfolge der Ventile ist gruppiert nach sechs Zonen mit je vier Ventilen: 1. Pfirsich 2. Stachelbeere 3. Maulbeere 4. Felsenbirne 5. Maibeere 6. Johannisbeere Der Index folgt dem Schema `z * 4 + v`, also vier Ventile pro Zone. ## Schnittstelle | Variable | Richtung | Bedeutung | |---|---:|---| | `xEnable` | Eingang | Freigabe fuer diese Betriebsart. Ist `xEnable = FALSE`, verlaesst der Baustein den Ablauf sofort mit `RETURN`. | | `bModeBit` | Eingang | Bitmaske dieser Betriebsart im Ventilstatus, im Handbetrieb standardmaessig `1`. | | `axValve` | Ausgang | Ventilmuster des Handbetriebs, Index `0..23`. | | `axLed` | Ausgang | Lampenmuster des Handbetriebs, Index `0..23`. | Wichtig: Bei `xEnable = FALSE` werden die Flipflops und Ausgangsmuster in diesem Baustein nicht neu berechnet. Die Instanz behaelt dadurch ihre bisherige Anwahl. ## Bedienlogik Jedes Ventil besitzt eine eigene `JK_FF`-Instanz in `fbJk[0..23]`. Der entprellte Tastendruck toggelt die Anwahl: - `J := TRUE` - `K := TRUE` - `Q` ist die gespeicherte Anwahl des Ventils - `tDebounce := T#20ms` wird an jede Instanz uebergeben Die lokalen Ausgaenge folgen direkt dem Flipflop-Zustand: ```st axValve[i] := fbJk[i].Q; axLed[i] := fbJk[i].Q; ``` ## Tasterquellen Die Feldtaster kommen aus dem Anvil-Namensraum: - `Anvil.<Zone>.xT_1` - `Anvil.<Zone>.xT_2` - `Anvil.<Zone>.xT_3` - `Anvil.<Zone>.xT_4` Fuer die Ventile 2 und 3 je Zone gibt es zusaetzlich HMI-/Bellows-Taster. Diese werden logisch mit dem jeweiligen Feldtaster verodert: ```st Anvil.<Zone>.xT_2 OR Bellows.<Zone>.xT_2 Anvil.<Zone>.xT_3 OR Bellows.<Zone>.xT_3 ``` Fuer `xT_1` und `xT_4` gibt es auf der Bedienoberflaeche in diesem Baustein keine zusaetzlichen Bellows-Taster. ## Abwahl von aussen `FB_TERMINAL_OUT` kann das Bit dieser Betriebsart in `Bellows.Betrieb.astValveStatus[i].bMode` loeschen, wenn ein offenes Ventil faellt beziehungsweise die Vorwahl verbraucht ist. Steht das Flipflop noch auf `Q = TRUE`, aber das Modus-Bit fehlt im Status, setzt `FB_MANUAL` das zugehoerige Flipflop zurueck: ```st RESET := fbJk[i].Q AND ((Bellows.Betrieb.astValveStatus[i].bMode AND bModeBit) = 0) ``` Damit wird verhindert, dass die Statusschleife das Modus-Bit im naechsten Zyklus sofort wieder setzt. ## Statusschreibung Am Ende des Bausteins wird fuer alle 24 Ventile der Status im Bellows-Spiegel aktualisiert: - Wenn `axValve[i] = TRUE`, wird `bModeBit` in `Bellows.Betrieb.astValveStatus[i].bMode` gesetzt. - Wenn `axValve[i] = FALSE`, wird `bModeBit` dort geloescht. - Bei angewaehltem Ventil wird `liquidationPeriod := T#0s` geschrieben. Im Handbetrieb bedeutet `T#0s`: keine automatische Laufzeitbegrenzung durch diesen Baustein; das Ventil bleibt angewaehlt, bis der Bediener es abwaehlt oder die externe Logik die Vorwahl verbraucht. Ob ein angewaehltes Ventil tatsaechlich oeffnet, entscheidet nicht `FB_MANUAL`, sondern die nachgelagerte Arbitrierung beziehungsweise Ausgabe in `FB_TERMINAL_OUT`. *)
FUNCTION_BLOCK FB_MANUAL
  VAR
    fbJk : ARRAY[0..23] OF JK_FF;  (* Ein JK-Flipflop je Ventil, Index z*4+v. Der entprellte Tastendruck toggelt die Anwahl; Q ist das Ventilmuster. *)
    tDebounce : TIME := T#20ms;  (* Entprellzeit der Taster, an jedes JK_FF gereicht (tDebounce). *)
    i : INT;  (* Laufindex ueber die 24 Ventile. *)
  END_VAR
  VAR_INPUT
    xEnable : BOOL;
    bModeBit : BYTE := 1;  (* Das Bit dieser Betriebsart im Ventilstatus (1 Manuell, 2 One-Shot, 4 wiederkehrend, 8 Auto) — wie GVL.Betrieb.uModeActive. *)
  END_VAR
  VAR_OUTPUT
    axValve : ARRAY[0..23] OF BOOL;  (* Das Ventilmuster dieser Betriebsart, Index z*4+v. In PLC_PRG waehlt der CASE aus, welcher Modus seinen Ausgang in den Spiegel legt. *)
    axLed : ARRAY[0..23] OF BOOL;  (* Das Lampenmuster dieser Betriebsart, Index z*4+v. In PLC_PRG waehlt der CASE aus, welcher Modus seinen Ausgang in den Spiegel legt. *)
  END_VAR

            (* ============================================================================
   FB_MANUAL  —  Handbetrieb, Betriebsart 1
   ----------------------------------------------------------------------------
   Projekt : Ackersteuerung (SoLaWi-Acker Bewaesserung)
   Autor   : Joerg Bernau / Blacksmith
   Datum   : 2026-09-21
   ----------------------------------------------------------------------------
   Vier Anschluesse, mehr nicht:
        xEnable   Freigabe der Betriebsart
        bModeBit  das Bit dieser Betriebsart im Ventilstatus (1)
        axValve   Ventilmuster, Index z*4+v   (Ausgang)
        axLed     Lampenmuster, Index z*4+v   (Ausgang)

   ENABLE: der Baustein verlaesst sich in der ERSTEN Zeile selbst, wenn
   xEnable FALSE ist. PLC_PRG ruft ihn dafuer in JEDEM Zyklus. Bei FALSE
   friert die Instanz ein und behaelt ihre Anwahl.

   JE VENTIL EIN FLIPFLOP, 24 Instanzen in fbJk: Zustand und Entprellung
   brauchen je Ventil ein eigenes Gedaechtnis. Der entprellte Druck toggelt
   (J = K = TRUE), Q ist die Anwahl. Die Entprellzeit ist tDebounce
   (lokal, T#20ms) und wird jedem JK_FF gereicht.

   DIE ABWAHL VON AUSSEN: FB_TERMINAL_OUT loescht das Bit dieses Modus in
   bMode, wenn ein offenes Ventil faellt — die Vorwahl ist verbraucht. Steht
   Q noch, aber das Bit fehlt, wird das Flipflop zurueckgesetzt (RESET), sonst
   setzte die Schleife unten das Bit im naechsten Takt wieder.

   Der Taster kommt vom Acker (Anvil.<Zone>.xT_1..4). Wo die Bedienoberflaeche
   einen eigenen Taster hat — xT_2 und xT_3 je Zone —, ist er dazu verodert;
   fuer xT_1 und xT_4 gibt es auf dieser Seite keinen.

   STATUS JE VENTIL: Bellows.Betrieb.astValveStatus[i].bMode traegt je
   Betriebsart ein Bit. Am Ende setzt eine Schleife das Bit dieses Modus
   (bModeBit) nach dem Ventilmuster — gesetzt, wo das Ventil angewaehlt ist,
   geloescht sonst. Die anderen Bits gehoeren den anderen Modi. Die
   Laufdauer eines angewaehlten Ventils ist im Handbetrieb T#0s: unbegrenzt,
   bis der Bediener es abwaehlt. Ob es wirklich oeffnet, entscheidet die
   Arbitrierung in FB_TERMINAL_OUT (isOpen).

   Index z*4+v, Reihenfolge Pfirsich, Stachelbeere, Maulbeere, Felsenbirne,
   Maibeere, Johannisbeere.
   ============================================================================ *)

IF NOT xEnable THEN
    RETURN;
END_IF;

(* --- Pfirsich, Ventile 1..4 --- *)
fbJk[0](xButton := Anvil.Pfirsich.xT_1, J := TRUE, K := TRUE, RESET := fbJk[0].Q AND ((Bellows.Betrieb.astValveStatus[0].bMode AND bModeBit) = 0), tDebounce := tDebounce);
axValve[0] := fbJk[0].Q;  axLed[0] := fbJk[0].Q;
fbJk[1](xButton := Anvil.Pfirsich.xT_2 OR Bellows.Pfirsich.xT_2, J := TRUE, K := TRUE, RESET := fbJk[1].Q AND ((Bellows.Betrieb.astValveStatus[1].bMode AND bModeBit) = 0), tDebounce := tDebounce);
axValve[1] := fbJk[1].Q;  axLed[1] := fbJk[1].Q;
fbJk[2](xButton := Anvil.Pfirsich.xT_3 OR Bellows.Pfirsich.xT_3, J := TRUE, K := TRUE, RESET := fbJk[2].Q AND ((Bellows.Betrieb.astValveStatus[2].bMode AND bModeBit) = 0), tDebounce := tDebounce);
axValve[2] := fbJk[2].Q;  axLed[2] := fbJk[2].Q;
fbJk[3](xButton := Anvil.Pfirsich.xT_4, J := TRUE, K := TRUE, RESET := fbJk[3].Q AND ((Bellows.Betrieb.astValveStatus[3].bMode AND bModeBit) = 0), tDebounce := tDebounce);
axValve[3] := fbJk[3].Q;  axLed[3] := fbJk[3].Q;

(* --- Stachelbeere, Ventile 1..4 --- *)
fbJk[4](xButton := Anvil.Stachelbeere.xT_1, J := TRUE, K := TRUE, RESET := fbJk[4].Q AND ((Bellows.Betrieb.astValveStatus[4].bMode AND bModeBit) = 0), tDebounce := tDebounce);
axValve[4] := fbJk[4].Q;  axLed[4] := fbJk[4].Q;
fbJk[5](xButton := Anvil.Stachelbeere.xT_2 OR Bellows.Stachelbeere.xT_2, J := TRUE, K := TRUE, RESET := fbJk[5].Q AND ((Bellows.Betrieb.astValveStatus[5].bMode AND bModeBit) = 0), tDebounce := tDebounce);
axValve[5] := fbJk[5].Q;  axLed[5] := fbJk[5].Q;
fbJk[6](xButton := Anvil.Stachelbeere.xT_3 OR Bellows.Stachelbeere.xT_3, J := TRUE, K := TRUE, RESET := fbJk[6].Q AND ((Bellows.Betrieb.astValveStatus[6].bMode AND bModeBit) = 0), tDebounce := tDebounce);
axValve[6] := fbJk[6].Q;  axLed[6] := fbJk[6].Q;
fbJk[7](xButton := Anvil.Stachelbeere.xT_4, J := TRUE, K := TRUE, RESET := fbJk[7].Q AND ((Bellows.Betrieb.astValveStatus[7].bMode AND bModeBit) = 0), tDebounce := tDebounce);
axValve[7] := fbJk[7].Q;  axLed[7] := fbJk[7].Q;

(* --- Maulbeere, Ventile 1..4 --- *)
fbJk[8](xButton := Anvil.Maulbeere.xT_1, J := TRUE, K := TRUE, RESET := fbJk[8].Q AND ((Bellows.Betrieb.astValveStatus[8].bMode AND bModeBit) = 0), tDebounce := tDebounce);
axValve[8] := fbJk[8].Q;  axLed[8] := fbJk[8].Q;
fbJk[9](xButton := Anvil.Maulbeere.xT_2 OR Bellows.Maulbeere.xT_2, J := TRUE, K := TRUE, RESET := fbJk[9].Q AND ((Bellows.Betrieb.astValveStatus[9].bMode AND bModeBit) = 0), tDebounce := tDebounce);
axValve[9] := fbJk[9].Q;  axLed[9] := fbJk[9].Q;
fbJk[10](xButton := Anvil.Maulbeere.xT_3 OR Bellows.Maulbeere.xT_3, J := TRUE, K := TRUE, RESET := fbJk[10].Q AND ((Bellows.Betrieb.astValveStatus[10].bMode AND bModeBit) = 0), tDebounce := tDebounce);
axValve[10] := fbJk[10].Q;  axLed[10] := fbJk[10].Q;
fbJk[11](xButton := Anvil.Maulbeere.xT_4, J := TRUE, K := TRUE, RESET := fbJk[11].Q AND ((Bellows.Betrieb.astValveStatus[11].bMode AND bModeBit) = 0), tDebounce := tDebounce);
axValve[11] := fbJk[11].Q;  axLed[11] := fbJk[11].Q;

(* --- Felsenbirne, Ventile 1..4 --- *)
fbJk[12](xButton := Anvil.Felsenbirne.xT_1, J := TRUE, K := TRUE, RESET := fbJk[12].Q AND ((Bellows.Betrieb.astValveStatus[12].bMode AND bModeBit) = 0), tDebounce := tDebounce);
axValve[12] := fbJk[12].Q;  axLed[12] := fbJk[12].Q;
fbJk[13](xButton := Anvil.Felsenbirne.xT_2 OR Bellows.Felsenbirne.xT_2, J := TRUE, K := TRUE, RESET := fbJk[13].Q AND ((Bellows.Betrieb.astValveStatus[13].bMode AND bModeBit) = 0), tDebounce := tDebounce);
axValve[13] := fbJk[13].Q;  axLed[13] := fbJk[13].Q;
fbJk[14](xButton := Anvil.Felsenbirne.xT_3 OR Bellows.Felsenbirne.xT_3, J := TRUE, K := TRUE, RESET := fbJk[14].Q AND ((Bellows.Betrieb.astValveStatus[14].bMode AND bModeBit) = 0), tDebounce := tDebounce);
axValve[14] := fbJk[14].Q;  axLed[14] := fbJk[14].Q;
fbJk[15](xButton := Anvil.Felsenbirne.xT_4, J := TRUE, K := TRUE, RESET := fbJk[15].Q AND ((Bellows.Betrieb.astValveStatus[15].bMode AND bModeBit) = 0), tDebounce := tDebounce);
axValve[15] := fbJk[15].Q;  axLed[15] := fbJk[15].Q;

(* --- Maibeere, Ventile 1..4 --- *)
fbJk[16](xButton := Anvil.Maibeere.xT_1, J := TRUE, K := TRUE, RESET := fbJk[16].Q AND ((Bellows.Betrieb.astValveStatus[16].bMode AND bModeBit) = 0), tDebounce := tDebounce);
axValve[16] := fbJk[16].Q;  axLed[16] := fbJk[16].Q;
fbJk[17](xButton := Anvil.Maibeere.xT_2 OR Bellows.Maibeere.xT_2, J := TRUE, K := TRUE, RESET := fbJk[17].Q AND ((Bellows.Betrieb.astValveStatus[17].bMode AND bModeBit) = 0), tDebounce := tDebounce);
axValve[17] := fbJk[17].Q;  axLed[17] := fbJk[17].Q;
fbJk[18](xButton := Anvil.Maibeere.xT_3 OR Bellows.Maibeere.xT_3, J := TRUE, K := TRUE, RESET := fbJk[18].Q AND ((Bellows.Betrieb.astValveStatus[18].bMode AND bModeBit) = 0), tDebounce := tDebounce);
axValve[18] := fbJk[18].Q;  axLed[18] := fbJk[18].Q;
fbJk[19](xButton := Anvil.Maibeere.xT_4, J := TRUE, K := TRUE, RESET := fbJk[19].Q AND ((Bellows.Betrieb.astValveStatus[19].bMode AND bModeBit) = 0), tDebounce := tDebounce);
axValve[19] := fbJk[19].Q;  axLed[19] := fbJk[19].Q;

(* --- Johannisbeere, Ventile 1..4 --- *)
fbJk[20](xButton := Anvil.Johannisbeere.xT_1, J := TRUE, K := TRUE, RESET := fbJk[20].Q AND ((Bellows.Betrieb.astValveStatus[20].bMode AND bModeBit) = 0), tDebounce := tDebounce);
axValve[20] := fbJk[20].Q;  axLed[20] := fbJk[20].Q;
fbJk[21](xButton := Anvil.Johannisbeere.xT_2 OR Bellows.Johannisbeere.xT_2, J := TRUE, K := TRUE, RESET := fbJk[21].Q AND ((Bellows.Betrieb.astValveStatus[21].bMode AND bModeBit) = 0), tDebounce := tDebounce);
axValve[21] := fbJk[21].Q;  axLed[21] := fbJk[21].Q;
fbJk[22](xButton := Anvil.Johannisbeere.xT_3 OR Bellows.Johannisbeere.xT_3, J := TRUE, K := TRUE, RESET := fbJk[22].Q AND ((Bellows.Betrieb.astValveStatus[22].bMode AND bModeBit) = 0), tDebounce := tDebounce);
axValve[22] := fbJk[22].Q;  axLed[22] := fbJk[22].Q;
fbJk[23](xButton := Anvil.Johannisbeere.xT_4, J := TRUE, K := TRUE, RESET := fbJk[23].Q AND ((Bellows.Betrieb.astValveStatus[23].bMode AND bModeBit) = 0), tDebounce := tDebounce);
axValve[23] := fbJk[23].Q;  axLed[23] := fbJk[23].Q;

(* --- Status je Ventil: das Bit dieser Betriebsart nach dem Muster,
       Laufdauer unbegrenzt (T#0s) --- *)
FOR i := 0 TO 23 DO
    IF axValve[i] THEN
        Bellows.Betrieb.astValveStatus[i].bMode := Bellows.Betrieb.astValveStatus[i].bMode OR bModeBit;
        Bellows.Betrieb.astValveStatus[i].liquidationPeriod := T#0s;
    ELSE
        Bellows.Betrieb.astValveStatus[i].bMode := Bellows.Betrieb.astValveStatus[i].bMode AND NOT bModeBit;
    END_IF;
END_FOR;

          
END_FUNCTION_BLOCK

(* # FB_SCHEDULE — One-Shot (2) und wiederkehrend (4) Ein Baustein fuer beide zeitgesteuerten Betriebsarten; `PLC_PRG` ruft ihn zweimal (`fbOneShot` mit `bModeBit := 2`, `fbRecurring` mit `bModeBit := 4`). Nur die Instanz mit `xEnable = TRUE` arbeitet; die andere haelt ihre Timer an (IN FALSE, ET bleibt) und schreibt nichts Gemeinsames. - **Anwahl:** je Beet ein `JK_FF` (`fbJk[0..23]`, J = K = TRUE). Feldtaster `Anvil.<Zone>.xT_v` und HMI-Puls `Schrittkette.axSelToggle[i]` schalten gleichberechtigt um; Q ist `Betrieb.aValveJobs[i].xSelected`. Nicht persistent. - **Befehle** (je eine steigende Flanke, `artCmd`): Start, Stopp, Pause, Quittieren aus `Schrittkette`. - **Zustand** `Schrittkette.uRunState`: 0 Idle, 1 Running, 2 Paused, 3 Done. Start laedt jedes angewaehlte Beet mit `tDuration > 0` (`liquidationPeriod` = Rest = Dauer, Timer zurueck). - **Nachwahl/Abwahl im Lauf** (Running oder Paused, `axSelPrev`): die steigende Flanke der Anwahl laedt das Beet sofort nach, es reiht sich ein; die fallende beendet es (Rest 0). Ein fertiges Beet bleibt angewaehlt, ohne neue Flanke, und laeuft nicht ein zweites Mal. - **Timer:** je Beet ein `TONR` (`aTonr[0..23]`, pausierbar). IN = Running UND Rest > 0 UND Ventil wirklich offen (Freigabe aus `FB_TERMINAL_OUT`). Pause und Warten auf Freigabe halten ihn an. - **Restzeit:** `astValveStatus[i].remainingLiquidation` = PT − ET, bei Q 0. Die HMI liest sie dort direkt; sie ist NICHT persistent. Eine Kopie in die persistente Job-Liste (`aValveJobs[i].tRemaining`) schrieb im Lauf alle 5 s die Persistenzdatei und ist seit 29.09.2026 entfallen. - **Ausgaenge:** `axValve[i]`/`axLed[i]` = Running UND Rest > 0; danach das Bit der Betriebsart in `astValveStatus[i].bMode`. **Offen:** wiederkehrend wertet `uStartHour`, `uStartMin` und `Betrieb.bWeekMask` noch nicht aus (Wochenschaltuhr folgt). *)
FUNCTION_BLOCK FB_SCHEDULE
  VAR
    i : INT;  (* Laufindex ueber die 24 Ventile. *)
    fbJk : ARRAY[0..23] OF JK_FF;  (* Ein JK-Flipflop je Beet, Index z*4+v in der Reihenfolge von FB_TERMINAL_OUT. Gleichberechtigt schalten um: der Taster am Beet (Anvil.<Zone>.xT_v) und der HMI-Puls auf Schrittkette.axSelToggle[i] (Beet-Taster im Bild, Vorwahl-Haken im Dialog); J = K = TRUE. Q ist Betrieb.aValveJobs[i].xSelected. Nicht persistent: nach einem Neustart ist nichts angewaehlt. *)
    aTonr : ARRAY[0..23] OF TONR;  (* Lauf-Timer je Beet (TONR, pausierbar): IN = Lauf aktiv (uRunState 1), Beet noch nicht fertig und Ventil wirklich offen; PT = astValveStatus[i].liquidationPeriod. Pause, Warten auf Freigabe und Sperre lassen IN fallen, ET bleibt stehen. Start und Stopp setzen per RESET zurueck. *)
    artCmd : ARRAY[0..3] OF R_TRIG;  (* Flanken der HMI-Befehle aus Schrittkette: 0 = xStart, 1 = xStop, 2 = xPause, 3 = xAcknowledge. *)
    axSelPrev : ARRAY[0..23] OF BOOL;  (* Anwahl je Beet im vorigen Zyklus: steigende Flanke im Lauf/Pause laedt das Beet nach, fallende beendet es. *)
  END_VAR
  VAR_TEMP
    xAny : BOOL;  (* Hilfsmerker: beim Start mindestens ein Beet geladen; im Lauf mindestens ein Beet noch nicht fertig. *)
  END_VAR
  VAR_INPUT
    xEnable : BOOL;  (* Master-Enable der One-Shot-Zone. FALSE setzt alle Anwahl-Flipflops zurueck (RESET der JK_FFs) -> Anwahl faellt, kein Ventil. Wird in PLC_PRG nur im One-Shot-Modus (uMode=2) auf TRUE gerufen; in anderen Modi nicht aufgerufen -> Instanz-Zustand friert ein. *)
    bModeBit : BYTE := 2;  (* Das Bit dieser Betriebsart im Ventilstatus (2 One-Shot, 4 wiederkehrend) — der Baustein dient beiden, PLC_PRG sagt ihm, welche. *)
  END_VAR
  VAR_OUTPUT
    axValve : ARRAY[0..23] OF BOOL;  (* Das Ventilmuster dieser Betriebsart, Index z*4+v. In PLC_PRG waehlt der CASE aus. *)
    axLed : ARRAY[0..23] OF BOOL;  (* Das Lampenmuster dieser Betriebsart, Index z*4+v. In PLC_PRG waehlt der CASE aus. *)
  END_VAR

            (* ============================================================================
   FB_SCHEDULE  —  Einmal-Lauf (2) und wiederkehrend (4)
   ----------------------------------------------------------------------------
   Projekt : Ackersteuerung (SoLaWi-Acker Bewaesserung)
   Autor   : Joerg Bernau / Blacksmith
   Datum   : 2026-09-21 (leergeraeumt), Lauf 2026-09-28
   ----------------------------------------------------------------------------
   Vier Anschluesse, mehr nicht:
        xEnable   Freigabe der Betriebsart
        bModeBit  das Bit dieser Betriebsart im Ventilstatus (2 oder 4 —
                  der Baustein dient beiden, PLC_PRG sagt ihm, welche)
        axValve   Ventilmuster, Index z*4+v   (Ausgang)
        axLed     Lampenmuster, Index z*4+v   (Ausgang)

   Zwei Instanzen (fbOneShot, fbRecurring). Nur die freigegebene kommt
   hinter das RETURN; die gesperrte haelt nur ihre Timer an (IN FALSE,
   ET bleibt stehen) und schreibt nichts Gemeinsames.

   ANWAHL: Betrieb.aValveJobs[i].xSelected ist STATUS und gehoert der SPS.
   Gleichberechtigt schalten um: der Taster am Beet (Anvil.<Zone>.xT_v)
   und der HMI-Puls auf Schrittkette.axSelToggle[i] (Beet-Taster im Bild,
   Vorwahl-Haken im Dialog). Je Beet ein JK_FF, Q ist die Anwahl. Nicht
   persistent: nach einem Neustart ist nichts angewaehlt.
   Die Zuordnung Index -> Zone/Ventil gibt FB_TERMINAL_OUT vor:
   Pfirsich 0-3, Stachelbeere 4-7, Maulbeere 8-11, Felsenbirne 12-15,
   Maibeere 16-19, Johannisbeere 20-23 (Index z*4+v, v = Taster/Ventil-1).

   LAUF (Schrittkette.uRunState: 0 Idle, 1 Running, 2 Paused, 3 Done):
        Start       Idle/Done: jedes angewaehlte Beet mit Dauer > 0 wird
                    geladen (liquidationPeriod = Rest = tDuration, Timer
                    zurueck) -> Running.  Paused -> Running.
        Pause       Running <-> Paused. Pausiert faellt das Bit, die Ventile
                    schliessen, die Timer stehen.
        Stopp       jeder Rest 0, Timer zurueck -> Idle.
        Quittieren  Done -> Idle.
        Nachwahl    Running/Paused: ein Beet, das JETZT angewaehlt wird
                    (steigende Flanke der Anwahl), wird sofort geladen und
                    reiht sich ein. Ein fertiges Beet bleibt angewaehlt, ohne
                    neue Flanke — es laeuft nicht ein zweites Mal.
        Abwahl      Running/Paused: ein Beet, das abgewaehlt wird, endet
                    sofort (Rest 0, Timer zurueck, Ventil zu).
   Ein Beet zaehlt, solange Running, Rest > 0 und das Ventil wirklich offen
   ist (Freigabe aus FB_TERMINAL_OUT) — ein TONR je Beet, der bei Pause und
   Warten stehen bleibt. Rest = PT - ET; Q -> Rest 0. Sind alle fertig ->
   Done. Die HMI zeigt die Restzeit direkt aus
   Betrieb.astValveStatus[i].remainingLiquidation — NICHT persistent. Eine
   Kopie in die persistente Job-Liste schrieb im Lauf alle 5 s die
   Persistenzdatei (29.09.2026) und ist deshalb entfallen.

   Alle Felder je Ventil laufen 0..23 (Index z*4+v).
   ============================================================================ *)

IF NOT xEnable THEN
    FOR i := 0 TO 23 DO
        aTonr[i](IN := FALSE, PT := Bellows.Betrieb.astValveStatus[i].liquidationPeriod, RESET := FALSE);
    END_FOR;
    RETURN;
END_IF;

(* --- 1) Anwahl je Beet: Feldtaster ODER HMI-Puls toggelt, Q ist der Status.
       Reihenfolge wie FB_TERMINAL_OUT. --- *)
(* Pfirsich: 0..3 *)
fbJk[0](xButton := Anvil.Pfirsich.xT_1 OR Bellows.Schrittkette.axSelToggle[0], J := TRUE, K := TRUE, RESET := FALSE, tDebounce := T#20ms);
fbJk[1](xButton := Anvil.Pfirsich.xT_2 OR Bellows.Schrittkette.axSelToggle[1], J := TRUE, K := TRUE, RESET := FALSE, tDebounce := T#20ms);
fbJk[2](xButton := Anvil.Pfirsich.xT_3 OR Bellows.Schrittkette.axSelToggle[2], J := TRUE, K := TRUE, RESET := FALSE, tDebounce := T#20ms);
fbJk[3](xButton := Anvil.Pfirsich.xT_4 OR Bellows.Schrittkette.axSelToggle[3], J := TRUE, K := TRUE, RESET := FALSE, tDebounce := T#20ms);
(* Stachelbeere: 4..7 *)
fbJk[4](xButton := Anvil.Stachelbeere.xT_1 OR Bellows.Schrittkette.axSelToggle[4], J := TRUE, K := TRUE, RESET := FALSE, tDebounce := T#20ms);
fbJk[5](xButton := Anvil.Stachelbeere.xT_2 OR Bellows.Schrittkette.axSelToggle[5], J := TRUE, K := TRUE, RESET := FALSE, tDebounce := T#20ms);
fbJk[6](xButton := Anvil.Stachelbeere.xT_3 OR Bellows.Schrittkette.axSelToggle[6], J := TRUE, K := TRUE, RESET := FALSE, tDebounce := T#20ms);
fbJk[7](xButton := Anvil.Stachelbeere.xT_4 OR Bellows.Schrittkette.axSelToggle[7], J := TRUE, K := TRUE, RESET := FALSE, tDebounce := T#20ms);
(* Maulbeere: 8..11 *)
fbJk[8](xButton := Anvil.Maulbeere.xT_1 OR Bellows.Schrittkette.axSelToggle[8], J := TRUE, K := TRUE, RESET := FALSE, tDebounce := T#20ms);
fbJk[9](xButton := Anvil.Maulbeere.xT_2 OR Bellows.Schrittkette.axSelToggle[9], J := TRUE, K := TRUE, RESET := FALSE, tDebounce := T#20ms);
fbJk[10](xButton := Anvil.Maulbeere.xT_3 OR Bellows.Schrittkette.axSelToggle[10], J := TRUE, K := TRUE, RESET := FALSE, tDebounce := T#20ms);
fbJk[11](xButton := Anvil.Maulbeere.xT_4 OR Bellows.Schrittkette.axSelToggle[11], J := TRUE, K := TRUE, RESET := FALSE, tDebounce := T#20ms);
(* Felsenbirne: 12..15 *)
fbJk[12](xButton := Anvil.Felsenbirne.xT_1 OR Bellows.Schrittkette.axSelToggle[12], J := TRUE, K := TRUE, RESET := FALSE, tDebounce := T#20ms);
fbJk[13](xButton := Anvil.Felsenbirne.xT_2 OR Bellows.Schrittkette.axSelToggle[13], J := TRUE, K := TRUE, RESET := FALSE, tDebounce := T#20ms);
fbJk[14](xButton := Anvil.Felsenbirne.xT_3 OR Bellows.Schrittkette.axSelToggle[14], J := TRUE, K := TRUE, RESET := FALSE, tDebounce := T#20ms);
fbJk[15](xButton := Anvil.Felsenbirne.xT_4 OR Bellows.Schrittkette.axSelToggle[15], J := TRUE, K := TRUE, RESET := FALSE, tDebounce := T#20ms);
(* Maibeere: 16..19 *)
fbJk[16](xButton := Anvil.Maibeere.xT_1 OR Bellows.Schrittkette.axSelToggle[16], J := TRUE, K := TRUE, RESET := FALSE, tDebounce := T#20ms);
fbJk[17](xButton := Anvil.Maibeere.xT_2 OR Bellows.Schrittkette.axSelToggle[17], J := TRUE, K := TRUE, RESET := FALSE, tDebounce := T#20ms);
fbJk[18](xButton := Anvil.Maibeere.xT_3 OR Bellows.Schrittkette.axSelToggle[18], J := TRUE, K := TRUE, RESET := FALSE, tDebounce := T#20ms);
fbJk[19](xButton := Anvil.Maibeere.xT_4 OR Bellows.Schrittkette.axSelToggle[19], J := TRUE, K := TRUE, RESET := FALSE, tDebounce := T#20ms);
(* Johannisbeere: 20..23 *)
fbJk[20](xButton := Anvil.Johannisbeere.xT_1 OR Bellows.Schrittkette.axSelToggle[20], J := TRUE, K := TRUE, RESET := FALSE, tDebounce := T#20ms);
fbJk[21](xButton := Anvil.Johannisbeere.xT_2 OR Bellows.Schrittkette.axSelToggle[21], J := TRUE, K := TRUE, RESET := FALSE, tDebounce := T#20ms);
fbJk[22](xButton := Anvil.Johannisbeere.xT_3 OR Bellows.Schrittkette.axSelToggle[22], J := TRUE, K := TRUE, RESET := FALSE, tDebounce := T#20ms);
fbJk[23](xButton := Anvil.Johannisbeere.xT_4 OR Bellows.Schrittkette.axSelToggle[23], J := TRUE, K := TRUE, RESET := FALSE, tDebounce := T#20ms);

FOR i := 0 TO 23 DO
    Bellows.Betrieb.aValveJobs[i].xSelected := fbJk[i].Q;
    (* Nachwahl und Abwahl waehrend des Laufs: die FLANKE der Anwahl, nicht
       ihr Zustand — ein fertiges Beet bleibt angewaehlt und laeuft nicht
       nochmal. Start laedt weiterhin alle Angewaehlten (Abschnitt 2). *)
    IF (Bellows.Schrittkette.uRunState = 1) OR (Bellows.Schrittkette.uRunState = 2) THEN
        IF fbJk[i].Q AND NOT axSelPrev[i]
           AND (Bellows.Betrieb.aValveJobs[i].tDuration > T#0s) THEN
            Bellows.Betrieb.astValveStatus[i].liquidationPeriod := Bellows.Betrieb.aValveJobs[i].tDuration;
            Bellows.Betrieb.astValveStatus[i].remainingLiquidation := Bellows.Betrieb.aValveJobs[i].tDuration;
            aTonr[i](IN := FALSE, PT := Bellows.Betrieb.aValveJobs[i].tDuration, RESET := TRUE);
        ELSIF NOT fbJk[i].Q AND axSelPrev[i] THEN
            Bellows.Betrieb.astValveStatus[i].remainingLiquidation := T#0s;
            aTonr[i](IN := FALSE, PT := Bellows.Betrieb.astValveStatus[i].liquidationPeriod, RESET := TRUE);
        END_IF;
    END_IF;
    axSelPrev[i] := fbJk[i].Q;
END_FOR;

(* --- 2) Befehle: je eine steigende Flanke --- *)
artCmd[0](CLK := Bellows.Schrittkette.xStart);
artCmd[1](CLK := Bellows.Schrittkette.xStop);
artCmd[2](CLK := Bellows.Schrittkette.xPause);
artCmd[3](CLK := Bellows.Schrittkette.xAcknowledge);

IF artCmd[1].Q THEN
    FOR i := 0 TO 23 DO
        Bellows.Betrieb.astValveStatus[i].remainingLiquidation := T#0s;
        aTonr[i](IN := FALSE, PT := Bellows.Betrieb.astValveStatus[i].liquidationPeriod, RESET := TRUE);
    END_FOR;
    Bellows.Schrittkette.uRunState := 0;
ELSIF artCmd[0].Q THEN
    IF Bellows.Schrittkette.uRunState = 2 THEN
        Bellows.Schrittkette.uRunState := 1;
    ELSIF Bellows.Schrittkette.uRunState <> 1 THEN
        xAny := FALSE;
        FOR i := 0 TO 23 DO
            IF Bellows.Betrieb.aValveJobs[i].xSelected
               AND (Bellows.Betrieb.aValveJobs[i].tDuration > T#0s) THEN
                Bellows.Betrieb.astValveStatus[i].liquidationPeriod := Bellows.Betrieb.aValveJobs[i].tDuration;
                Bellows.Betrieb.astValveStatus[i].remainingLiquidation := Bellows.Betrieb.aValveJobs[i].tDuration;
                aTonr[i](IN := FALSE, PT := Bellows.Betrieb.aValveJobs[i].tDuration, RESET := TRUE);
                xAny := TRUE;
            END_IF;
        END_FOR;
        IF xAny THEN
            Bellows.Schrittkette.uRunState := 1;
        END_IF;
    END_IF;
ELSIF artCmd[2].Q THEN
    IF Bellows.Schrittkette.uRunState = 1 THEN
        Bellows.Schrittkette.uRunState := 2;
    ELSIF Bellows.Schrittkette.uRunState = 2 THEN
        Bellows.Schrittkette.uRunState := 1;
    END_IF;
ELSIF artCmd[3].Q AND (Bellows.Schrittkette.uRunState = 3) THEN
    Bellows.Schrittkette.uRunState := 0;
END_IF;

(* --- 3) Lauf je Beet: Timer, Restzeit, Muster --- *)
xAny := FALSE;
FOR i := 0 TO 23 DO
    aTonr[i](IN := (Bellows.Schrittkette.uRunState = 1)
                   AND (Bellows.Betrieb.astValveStatus[i].remainingLiquidation > T#0s)
                   AND Bellows.Betrieb.astValveStatus[i].isOpen,
             PT := Bellows.Betrieb.astValveStatus[i].liquidationPeriod,
             RESET := FALSE);

    IF Bellows.Betrieb.astValveStatus[i].remainingLiquidation > T#0s THEN
        IF aTonr[i].Q THEN
            Bellows.Betrieb.astValveStatus[i].remainingLiquidation := T#0s;
        ELSE
            Bellows.Betrieb.astValveStatus[i].remainingLiquidation :=
                Bellows.Betrieb.astValveStatus[i].liquidationPeriod - aTonr[i].ET;
        END_IF;
    END_IF;

    axValve[i] := (Bellows.Schrittkette.uRunState = 1)
                  AND (Bellows.Betrieb.astValveStatus[i].remainingLiquidation > T#0s);
    axLed[i] := axValve[i];
    xAny := xAny OR (Bellows.Betrieb.astValveStatus[i].remainingLiquidation > T#0s);
END_FOR;

IF (Bellows.Schrittkette.uRunState = 1) AND NOT xAny THEN
    Bellows.Schrittkette.uRunState := 3;
END_IF;

(* --- 4) Status je Ventil: das Bit dieser Betriebsart nach dem Muster --- *)
FOR i := 0 TO 23 DO
    IF axValve[i] THEN
        Bellows.Betrieb.astValveStatus[i].bMode := Bellows.Betrieb.astValveStatus[i].bMode OR bModeBit;
    ELSE
        Bellows.Betrieb.astValveStatus[i].bMode := Bellows.Betrieb.astValveStatus[i].bMode AND NOT bModeBit;
    END_IF;
END_FOR;

          
END_FUNCTION_BLOCK

(* # FB_WEEKLY_TIMER — Zeitbasis / Wochenplan Liest die UNIX-Echtzeit über `FB_SYS_TIME`, zerlegt sie per **Hinnant-Civil-Date** in die DUT `ST_DateTime` (`dtNow`, struct-tm-Stil, UTC) und bildet ein Wochenplan-Fenster: `xWtQ`=TRUE wenn Wochentag in `bWtDays` (`T_WeekMask`, Mo..So) freigegeben UND Uhrzeit im Fenster `[Start,End)` (mitternachtsübergreifend). `dtNow` ist Output + wird von `FB_MANUAL_TIME` für den Startzeit-Vergleich je Job genutzt. *)
FUNCTION_BLOCK FB_WEEKLY_TIMER
  VAR
    i : INT;  (* Laufindex ueber die 24 Ventile. *)
  END_VAR
  VAR_INPUT
    xEnable : BOOL;  (* Freigabe der Betriebsart. FALSE = der Baustein verlaesst sich in seiner ersten Zeile und schreibt nichts in die Spiegel — der aktive Modus bleibt unangetastet. *)
    bModeBit : BYTE := 8;  (* Das Bit dieser Betriebsart im Ventilstatus (8 Auto). *)
  END_VAR
  VAR_OUTPUT
    axValve : ARRAY[0..23] OF BOOL;  (* Das Ventilmuster dieser Betriebsart, Index z*4+v. In PLC_PRG waehlt der CASE aus. *)
    axLed : ARRAY[0..23] OF BOOL;  (* Das Lampenmuster dieser Betriebsart, Index z*4+v. In PLC_PRG waehlt der CASE aus. *)
  END_VAR

            (* ============================================================================
   FB_WEEKLY_TIMER  —  Auto, Betriebsart 8
   ----------------------------------------------------------------------------
   Projekt : Ackersteuerung (SoLaWi-Acker Bewaesserung)
   Autor   : Joerg Bernau / Blacksmith
   Datum   : 2026-09-21 (leergeraeumt fuer den Neuaufbau)
   ----------------------------------------------------------------------------
   Vier Anschluesse, mehr nicht:
        xEnable   Freigabe der Betriebsart
        bModeBit  das Bit dieser Betriebsart im Ventilstatus (8)
        axValve   Ventilmuster, Index z*4+v   (Ausgang)
        axLed     Lampenmuster, Index z*4+v   (Ausgang)

   ENABLE: der Baustein verlaesst sich in der ERSTEN Zeile selbst, wenn
   xEnable FALSE ist. PLC_PRG ruft ihn dafuer in JEDEM Zyklus. Bei FALSE
   friert die Instanz ein.

   STATUS JE VENTIL: Bellows.Betrieb.astValveStatus[i].bMode traegt je
   Betriebsart ein Bit; die Schleife am Ende setzt das Bit dieses Modus
   nach dem Ventilmuster.

   Der Rumpf ist leer und wird Schritt fuer Schritt neu gebaut. Die alte
   Kalenderrechnung ist mit ihren Datentypen (ST_DateTime, T_WeekMask,
   ST_TimerConfig) entfallen.
   ============================================================================ *)

IF NOT xEnable THEN
    RETURN;
END_IF;

(* --- Status je Ventil: das Bit dieser Betriebsart nach dem Muster --- *)
FOR i := 0 TO 23 DO
    IF axValve[i] THEN
        Bellows.Betrieb.astValveStatus[i].bMode := Bellows.Betrieb.astValveStatus[i].bMode OR bModeBit;
    ELSE
        Bellows.Betrieb.astValveStatus[i].bMode := Bellows.Betrieb.astValveStatus[i].bMode AND NOT bModeBit;
    END_IF;
END_FOR;

          
END_FUNCTION_BLOCK

(* # PLC_PRG — Hauptprogramm Ackersteuerung `PLC_PRG` ist das zyklische Hauptprogramm der Ackersteuerung. Es ruft die Betriebsarten-Bausteine in jedem SPS-Zyklus auf und uebergibt jedem Baustein seine Freigabe ueber `xEnable` sowie das zugehoerige Modus-Bit ueber `bModeBit`. Die aktuell aktive Betriebsart kommt aus `GVL.Betrieb.uModeActive`: | Wert | Betriebsart | Baustein | |---:|---|---| | `0` | AUS | keine Vorwahl aktiv, Ausgabe faellt ab | | `1` | Manuell | `FB_MANUAL` | | `2` | Einmal-Lauf / One-Shot | `FB_SCHEDULE` | | `4` | Wiederkehrend | `FB_SCHEDULE` | | `8` | Auto | `FB_WEEKLY_TIMER` | ## Zyklischer Ablauf 1. `fbManual` wird mit `xEnable := (GVL.Betrieb.uModeActive = 1)` aufgerufen. 2. `fbOneShot` wird mit `xEnable := (GVL.Betrieb.uModeActive = 2)` aufgerufen. 3. `fbRecurring` wird mit `xEnable := (GVL.Betrieb.uModeActive = 4)` aufgerufen. 4. `fbAuto` wird mit `xEnable := (GVL.Betrieb.uModeActive = 8)` aufgerufen. 5. `fbOut` wird als zentraler Ausgabe- und Arbitrierungsbaustein mit `xEnable := (GVL.Betrieb.uModeActive <> 0)` aufgerufen. Die Modus-Bausteine schreiben ihre Vorwahl je Ventil in `Bellows.Betrieb.astValveStatus[i].bMode`. Der zentrale Setter `FB_TERMINAL_OUT` liest daraus die Vorwahl der aktiven Betriebsart, arbitriert die gleichzeitig offenen Ventile und schreibt die realen Ventil- und LED-Ausgaenge. ## Architekturhinweis Es gibt keinen lokalen Ventilspiegel mehr im Hauptprogramm. Der gemeinsame Zustand je Ventil liegt in `Bellows.Betrieb.astValveStatus`. Damit ist `FB_TERMINAL_OUT` die zentrale Stelle fuer: - Vorwahl der aktiven Betriebsart - Begrenzung ueber `GVL.Betrieb.uMaxVentile` - reale Ventilausgaenge `Anvil.<Zone>.xV_1..4` - LED-Ausgaenge `Anvil.<Zone>.xLed_5..8` Bei Betriebsart `0` wird `fbOut` deaktiviert; der Ausgabe-Baustein laesst dann alle Freigaben und Klemmen abfallen. *)
PROGRAM PLC_PRG
  VAR
    fbOut : FB_TERMINAL_OUT;  (* Der eine Sammler: Grant auf die Ventilklemmen, LED-Bild auf die Status-LEDs, einmal je Zyklus. *)
    fbManual : FB_MANUAL;  (* Betriebsart 1 — Manuell. Laeuft jeden Zyklus, xEnable entscheidet. *)
    fbOneShot : FB_SCHEDULE;  (* Betriebsart 2 — One-Shot-Schrittkette. Laeuft jeden Zyklus, xEnable entscheidet. *)
    fbRecurring : FB_SCHEDULE;  (* Betriebsart 4 — wiederkehrend (Zeit-Scheduler, Wochentag-gated). Laeuft jeden Zyklus, xEnable entscheidet. *)
    fbAuto : FB_WEEKLY_TIMER;  (* Betriebsart 8 — Auto. Laeuft jeden Zyklus, xEnable entscheidet. Typ vorlaeufig FB_WEEKLY_TIMER, der einzige Modus-Baustein ohne Aufrufer. *)
  END_VAR

            (* ============================================================================
   PLC_PRG  —  Hauptprogramm Ackersteuerung (SoLaWi-Acker Bewaesserung)
   ----------------------------------------------------------------------------
   Neuaufbau 2026-09-21/22: die Betriebsart liefert, die DUT traegt, der
   Setter entscheidet.

   Die vier Modus-Bausteine sind UNTERPROGRAMME: jeder wird in JEDEM Zyklus
   gerufen, und sein xEnable entscheidet, ob er arbeitet. Ein abgeschalteter
   Baustein verlaesst sich in seiner ersten Zeile selbst und friert ein — der
   Lauf geht weiter, wo er stand, sobald der Bediener zurueckkommt.

   Die Betriebsart ist GVL.Betrieb.uModeActive, die EINE Quelle, ohne lokale
   Kopie, je Betriebsart ein Bit:
        1 = Manuell · 2 = One-Shot · 4 = wiederkehrend · 8 = Auto · 0 = AUS
   Dasselbe Bit bekommt jeder Baustein als bModeBit und setzt es je Ventil
   in Bellows.Betrieb.astValveStatus[i].bMode — der Status ueber die Modi.

   KEIN SPIEGEL MEHR: der Zustand je Ventil steht in der DUT
   (Bellows.Betrieb.astValveStatus). FB_TERMINAL_OUT liest daraus die
   Vorwahl der aktiven Betriebsart, arbitriert (uMaxVentile; die Vorwahl
   verbraucht sich mit dem Lauf) und legt Freigabe und Lampen auf
   die 48 Klemmen. Ein Modus, der nicht aktiv ist, wird gar nicht gelesen —
   ein CASE, der sein eingefrorenes Muster auswaehlte, ist damit entfallen.
   ============================================================================ *)

(* --- 1) Die vier Betriebsarten. Nur eine arbeitet, alle werden gerufen. --- *)
fbManual(xEnable := (GVL.Betrieb.uModeActive = 1), bModeBit := 1);
fbOneShot(xEnable := (GVL.Betrieb.uModeActive = 2), bModeBit := 2);
fbRecurring(xEnable := (GVL.Betrieb.uModeActive = 4), bModeBit := 4);
fbAuto(xEnable := (GVL.Betrieb.uModeActive = 8), bModeBit := 8);

(* --- 2) Ausgabe: der eine Setter, Arbitrierung auf der DUT, 48 Klemmen.
       AUS heisst: nichts vorgewaehlt, alles faellt. --- *)
fbOut(xEnable := (GVL.Betrieb.uModeActive <> 0));

(* --- Sonde (Debug): HMI-Taster direkt auf das Ventil, am Modus vorbei. --- *)
//Anvil.Stachelbeere.xV_2 := Bellows.Stachelbeere.xT_2;
//Anvil.Stachelbeere.xV_3 := Bellows.Stachelbeere.xT_3;

          
END_PROGRAM

(* # FC_GetKcValue — FAO-56 Kc-Pflanzenkoeffizient (Phase-4-Modell) Liefert den Pflanzenkoeffizienten Kc für den Kultur-Tag `iDay_crop` aus der Kurve `ST_KcCurve` (FAO-56): Initial konstant → Development linear `kc_initial→kc_mid` → Mid-Season konstant → Late linear `kc_mid→kc_end` → danach 0. Wasserbedarf **ETc = ET0 × Kc**. **Phase 4 zurückgestellt** — ET0-/Sensorik-Hardware (geplant per LoRaWAN) fehlt; Referenzmodell = Geisenheimer Steuerung (GSEHEN). *)
FUNCTION FC_GetKcValue : REAL
  VAR
    iDays_to_mid : INT;
    iDays_to_end : INT;
    rFrac : REAL;
  END_VAR
  VAR_INPUT
    stKcCurve : ST_KcCurve;
    iDay_crop : INT;
  END_VAR

            (* ============================================================================
   FC_GetKcValue  —  FAO-56 Kc-Pflanzenkoeffizient (Phase-4-Modell)
   ----------------------------------------------------------------------------
   Projekt : Ackersteuerung (SoLaWi-Acker Bewaesserung)
   Autor   : Joerg Bernau
   Datum   : 2026-06-05
   ----------------------------------------------------------------------------
   Zweck   : Liefert den Pflanzenkoeffizienten Kc fuer den Kultur-Tag iDay_crop
             aus der Kurve stKcCurve (FAO-56): Initial konstant; Development
             linear kc_initial->kc_mid; Mid-Season konstant kc_mid; Late linear
             kc_mid->kc_end; danach 0. Wasserbedarf ETc = ET0 * Kc.
   ============================================================================ *)

iDays_to_mid := stKcCurve.days_initial + stKcCurve.days_dev;
iDays_to_end := iDays_to_mid + stKcCurve.days_mid + stKcCurve.days_late;

IF iDay_crop <= stKcCurve.days_initial THEN
    FC_GetKcValue := stKcCurve.kc_initial;

ELSIF iDay_crop <= stKcCurve.days_initial + stKcCurve.days_dev THEN
    rFrac := REAL(iDay_crop - stKcCurve.days_initial) / REAL(stKcCurve.days_dev);
    FC_GetKcValue := stKcCurve.kc_initial + rFrac * (stKcCurve.kc_mid - stKcCurve.kc_initial);

ELSIF iDay_crop <= iDays_to_mid + stKcCurve.days_mid THEN
    FC_GetKcValue := stKcCurve.kc_mid;

ELSIF iDay_crop <= iDays_to_end THEN
    rFrac := REAL(iDay_crop - (iDays_to_mid + stKcCurve.days_mid)) / REAL(stKcCurve.days_late);
    FC_GetKcValue := stKcCurve.kc_mid + rFrac * (stKcCurve.kc_end - stKcCurve.kc_mid);

ELSE
    FC_GetKcValue := 0.0;
END_IF;
          
END_FUNCTION

(* Koppler im Schaltschrank (Weidmueller UR20-FBC-MOD-TCP, 192.168.24.229, Segment MODBUS_NORD) mit 8 digitalen Ein- und 8 Ausgaengen DI_0..7 und DO_0..7. Derzeit vom Programm nicht verwendet; die Betriebsart kommt aus der HMI-Gruppe Betrieb, nicht mehr von einem Wahlschalter. *)
PROGRAM Schaltschrank
  VAR_GLOBAL
    DI_0 AT %IX6.0 : BOOL;
    DI_1 AT %IX6.1 : BOOL;
    DI_2 AT %IX6.2 : BOOL;
    DI_3 AT %IX6.3 : BOOL;
    DI_4 AT %IX6.4 : BOOL;
    DI_5 AT %IX6.5 : BOOL;
    DI_6 AT %IX6.6 : BOOL;
    DI_7 AT %IX6.7 : BOOL;
    DO_0 AT %QX6.0 : BOOL;
    DO_1 AT %QX6.1 : BOOL;
    DO_2 AT %QX6.2 : BOOL;
    DO_3 AT %QX6.3 : BOOL;
    DO_4 AT %QX6.4 : BOOL;
    DO_5 AT %QX6.5 : BOOL;
    DO_6 AT %QX6.6 : BOOL;
    DO_7 AT %QX6.7 : BOOL;
  END_VAR

            
          
END_PROGRAM

(* # FB_DEVICE_MONITOR — Geräte-/Modul-Zustandsgraph + Klartext Überwacht den Comm-Status EINES Geräts/Moduls. Zustandsgraph `uDmState`: **0 Unbekannt → 1 Online → 2 Gestört → 3 Offline** (entprellt über `tDmFault`/`tDmRecover`). Eingänge `xStatusValid` (Quelle liefert Daten) + `xOnline` (Gerät antwortet). Ausgabe: `uDmState` + **Klartext-STRING** `sDmStatus` (`Online`/`Gestört`/`Keine Verbindung`/`Unbekannt`/`Status-Quelle fehlt`). **Quellen-agnostisch** — passt auf Modbus-Comm-Status UND LoRaWAN-Uplink-Liveness. *)
FUNCTION_BLOCK FB_DEVICE_MONITOR
  VAR
    tonDmFault : TON;  (* Entprell-Timer Offline *)
    tonDmRecover : TON;  (* Entprell-Timer Wiederkehr (stabil online) *)
  END_VAR
  VAR_INPUT
    xStatusValid : BOOL;  (* Status-Quelle liefert Daten; FALSE = Quelle fehlt -> Zustand Unbekannt *)
    xOnline : BOOL;  (* Geraet antwortet (Modbus-Transaktion ok); nur gueltig bei xStatusValid *)
    tDmFault : TIME := T#3S;  (* Entprellung: Dauer ohne Antwort bis OFFLINE *)
    tDmRecover : TIME := T#2S;  (* Dauer stabil online bis wieder ONLINE *)
  END_VAR
  VAR_OUTPUT
    uDmState : USINT;  (* Zustand: 0=Unbekannt, 1=Online, 2=Gestoert, 3=Offline *)
    sDmStatus : STRING;  (* Klartext-Status fuer die HMI *)
  END_VAR

            (* ============================================================================
   FB_DEVICE_MONITOR  —  Geraete-/Modulueberwachung mit Zustandsgraph + Klartext
   ----------------------------------------------------------------------------
   Projekt : Ackersteuerung (SoLaWi-Acker Bewaesserung)
   Autor   : Joerg Bernau / Blacksmith
   Datum   : 2026-06-06
   ----------------------------------------------------------------------------
   Zweck   : Ueberwacht den Comm-Status EINES Modbus-Geraets (bzw. Moduls) und
             liefert einen entprellten Zustand + einen KLARTEXT-STRING fuer die
             HMI (die rohen Status-Bits werden nicht an die HMI durchgereicht).
             Eingang xOnline kommt aus dem Runtime-Comm-Status (sobald verfuegbar);
             xStatusValid=FALSE => Quelle fehlt => Zustand Unbekannt.

   Zustandsgraph (uDmState):
     0 Unbekannt --(Quelle gueltig)--> Online (xOnline) | Offline (sonst)
     1 Online    --(kurzer Aussetzer)--> Gestoert
                 --(Offline laenger als tDmFault)--> Offline
     2 Gestoert  --(stabil online tDmRecover)--> Online
                 --(Offline laenger als tDmFault)--> Offline
     3 Offline   --(stabil online tDmRecover)--> Online
   HINWEIS : KEIN RETURN — der cxx-Transpiler kennt RETURN noch nicht. Der
             "Quelle fehlt"-Zweig laeuft daher als IF/ELSE (kein early-exit).
   ============================================================================ *)

(* --- Ohne gueltige Quelle: Unbekannt, Timer ruhen --- *)
IF NOT xStatusValid THEN
    uDmState  := 0;
    sDmStatus := 'Status-Quelle fehlt';
    tonDmFault(IN := FALSE, PT := tDmFault);
    tonDmRecover(IN := FALSE, PT := tDmRecover);
ELSE
    (* --- Entprell-Timer --- *)
    tonDmFault(IN := NOT xOnline, PT := tDmFault);
    tonDmRecover(IN := xOnline, PT := tDmRecover);

    (* --- Zustandsgraph --- *)
    IF uDmState = 0 THEN
        IF xOnline THEN uDmState := 1; ELSE uDmState := 3; END_IF;
    ELSIF NOT xOnline THEN
        IF tonDmFault.Q THEN
            uDmState := 3;                 (* dauerhaft weg -> Offline *)
        ELSIF uDmState = 1 THEN
            uDmState := 2;                 (* kurzer Aussetzer -> Gestoert *)
        END_IF;
    ELSE
        IF tonDmRecover.Q THEN
            uDmState := 1;                 (* stabil zurueck -> Online *)
        END_IF;
    END_IF;

    (* --- Klartext fuer die HMI --- *)
    IF    uDmState = 1 THEN sDmStatus := 'Online';
    ELSIF uDmState = 2 THEN sDmStatus := 'Gestoert';
    ELSIF uDmState = 3 THEN sDmStatus := 'Keine Verbindung';
    ELSE                    sDmStatus := 'Unbekannt';
    END_IF;
END_IF;
          
END_FUNCTION_BLOCK

(* # FB_BUS_MONITOR — Aggregierte Geräteüberwachung für die HMI Führt je Gerät eine `FB_DEVICE_MONITOR`-Instanz (7 Geräte) und bündelt: Zustand (`auBmState`) + Klartext (`asBmStatus`) je Gerät, Sammel-OK (`xBmAllOk`), Fehlerzahl (`iBmFaultCount`), Sammel-Klartext (`sBmSummary`). Eingänge: `xBmValid` + `axBmOnline[0..6]` (0=Pfirsich 1=Stachelbeere 2=Maulbeere 3=Felsenbirne 4=Maibeere 5=Johannisbeere 6=Schaltschrank), gespeist aus `Anvil.<grp>.Status.xOnline`. In PLC_PRG §9 → `Bellows.Diag.*` (HMI rendert Klartext aus dem Zustandscode). *)
FUNCTION_BLOCK FB_BUS_MONITOR
  VAR
    afbBmMon : ARRAY[0..6] OF FB_DEVICE_MONITOR;  (* Pro-Geraet-Zustandsgraph-Instanzen *)
    iBm : INT;  (* Schleifenindex 0..6 *)
  END_VAR
  VAR_INPUT
    xBmValid : BOOL;  (* Status-Quelle (Dev-Monitor / LoRaWAN-Netzserver) liefert Daten *)
    axBmOnline : ARRAY[0..6] OF BOOL;  (* Online je Geraet: 0=Pfirsich 1=Stachelbeere 2=Maulbeere 3=Felsenbirne 4=Maibeere 5=Johannisbeere 6=Schaltschrank *)
  END_VAR
  VAR_OUTPUT
    asBmStatus : ARRAY[0..6] OF STRING;  (* Klartext-Status je Geraet (fuer HMI) *)
    auBmState : ARRAY[0..6] OF USINT;  (* Zustand je Geraet (0=Unbekannt 1=Online 2=Gestoert 3=Offline) *)
    xBmAllOk : BOOL;  (* TRUE = alle Geraete online *)
    iBmFaultCount : INT;  (* Anzahl Geraete nicht online (Gestoert/Offline/Unbekannt) *)
    sBmSummary : STRING;  (* Sammel-Klartext fuer die HMI *)
  END_VAR

            (* ============================================================================
   FB_BUS_MONITOR  —  Aggregierte Geraete-/Modulueberwachung fuer die HMI
   ----------------------------------------------------------------------------
   Projekt : Ackersteuerung (SoLaWi-Acker Bewaesserung)
   Autor   : Joerg Bernau / Blacksmith
   Datum   : 2026-06-06
   ----------------------------------------------------------------------------
   Zweck   : Fuehrt je ueberwachtem Geraet eine FB_DEVICE_MONITOR-Instanz
             (Zustandsgraph + Klartext) und buendelt die Ergebnisse fuer die
             HMI: Klartext je Geraet (asBmStatus), Zustand je Geraet (auBmState),
             Sammel-OK (xBmAllOk), Fehlerzahl (iBmFaultCount) und eine
             Sammelmeldung (sBmSummary).
             Quelle der Online-Bits (axBmOnline) liefert die Runtime-Monitor-
             Schicht (Dev) bzw. der LoRaWAN-Netzserver (Uplink-Liveness). Bis
             dahin xBmValid=FALSE -> alle Geraete 'Status-Quelle fehlt'.
             Geraete-Index: 0=Pfirsich 1=Stachelbeere 2=Maulbeere 3=Felsenbirne
             4=Maibeere 5=Johannisbeere 6=Schaltschrank.
   ============================================================================ *)

xBmAllOk      := TRUE;
iBmFaultCount := 0;

FOR iBm := 0 TO 6 DO
    afbBmMon[iBm](xStatusValid := xBmValid, xOnline := axBmOnline[iBm]);
    auBmState[iBm]  := afbBmMon[iBm].uDmState;
    asBmStatus[iBm] := afbBmMon[iBm].sDmStatus;
    IF afbBmMon[iBm].uDmState <> 1 THEN          (* alles ausser Online = Stoerung *)
        xBmAllOk      := FALSE;
        iBmFaultCount := iBmFaultCount + 1;
    END_IF;
END_FOR;

(* --- Sammelmeldung (Klartext) fuer die HMI --- *)
IF NOT xBmValid THEN
    sBmSummary := 'Ueberwachung: Status-Quelle fehlt';
ELSIF xBmAllOk THEN
    sBmSummary := 'Alle Geraete online';
ELSE
    sBmSummary := 'Stoerung: Geraet(e) nicht online';
END_IF;
          
END_FUNCTION_BLOCK

(* HMI-Gruppe Diag: Geraeteueberwachung fuer die HMI. auDevState[0..6] Zustand je Geraet (0 Unbekannt, 1 Online, 2 Gestoert, 3 Keine Verbindung), asDevStatus und sSummary als Klartext, xAllOk und iFaultCount als Sammelmeldung. Index 0 Pfirsich, 1 Stachelbeere, 2 Maulbeere, 3 Felsenbirne, 4 Maibeere, 5 Johannisbeere, 6 Schaltschrank. *)
PROGRAM Diag
  VAR_GLOBAL
    asDevStatus AT %MD1 : ARRAY[0..6] OF STRING;  (* Klartext-Status je Geraet fuer HMI (0=Pfirsich..5=Johannisbeere,6=Schaltschrank) *)
    auDevState AT %MD2 : ARRAY[0..6] OF USINT;  (* Zustand je Geraet fuer HMI-Farbcodierung (0=Unbekannt 1=Online 2=Gestoert 3=Offline) *)
    sSummary AT %MD3 : STRING;  (* Sammel-Klartext der Geraeteueberwachung fuer HMI *)
    xAllOk AT %MX0.0 : BOOL;  (* TRUE = alle Geraete online (HMI-Sammelanzeige) *)
    iFaultCount AT %MW0 : INT;  (* Anzahl Geraete nicht online (HMI) *)
  END_VAR

            
          
END_PROGRAM

(* HMI-Gruppe HmiCmd: derzeit ohne Variablen. *)
PROGRAM HmiCmd

            
          
END_PROGRAM

(* Programm in taskDiag (200 ms): liest je Geraet den Online-Status aus Anvil.<Geraet>.Status, wertet ihn mit FB_BUS_MONITOR aus (Zustandsgraph mit Entprellung je Geraet) und schreibt das Ergebnis nach Bellows.Diag, damit die HMI es anzeigt. Die Geraete-Indizes sind handgepflegt (0 Pfirsich bis 6 Schaltschrank); ein neues Geraet muss hier und in FB_BUS_MONITOR nachgetragen werden. *)
PROGRAM BusMonitor
  VAR
    mon : FB_BUS_MONITOR;  (* Aggregierte Geraeteueberwachung *)
    axOnline : ARRAY[0..6] OF BOOL;  (* Online-Bits je Geraet, Index wie in FB_BUS_MONITOR *)
  END_VAR

            (* ============================================================================
   BusMonitor  -  Runtime-Comm-Status  ->  FB_BUS_MONITOR  ->  Bellows/Hearth
   ----------------------------------------------------------------------------
   Drei Glieder, von denen bis heute nur das mittlere existierte:

   1. QUELLE  Der cxx-Codegen materialisiert je Anvil-Geraetegruppe eine
              read-only Status-Sub-Struct unter Anvil.<grp>.Status , gefuellt
              im Input-Scan VOR der POU-Ausfuehrung - pro Zyklus ein
              konsistentes Abbild. Vertrag:
              documentation/architecture/device-status-interface.md

   2. LOGIK   FB_BUS_MONITOR fuehrt je Geraet eine FB_DEVICE_MONITOR-Instanz
              (Zustandsgraph, Entprellung, Klartext) und buendelt sie. Steht
              seit 2026-06-06, lief aber mit xBmValid=FALSE leer, weil
              axBmOnline keinen Lieferanten hatte.

   3. SENKE   Der Deskriptor kennt nur POOL-Variablen mit bellowsRead. Was in
              der FB-Instanz bleibt, sieht Hearth nie. Die Bellows.Diag-
              Variablen sind dafuer angelegt und tragen die Flagge bereits -
              es fehlten nur die fuenf Zuweisungen unten.

   Index-Zuordnung wie in FB_BUS_MONITOR dokumentiert:
     0=Pfirsich 1=Stachelbeere 2=Maulbeere 3=Felsenbirne
     4=Maibeere 5=Johannisbeere 6=Schaltschrank

   ACHTUNG: Die Zuordnung ist HANDGEPFLEGT und an ARRAY[0..6] gebunden. Ein
   achtes Geraet bliebe unueberwacht, ein geloeschtes verschoebe alle
   folgenden Indizes - die HMI meldete dann das falsche Geraet. Der
   Automatismus, der das aus der Bus-Topologie ableitet, ist offen.
   ============================================================================ *)

(* --- 1. Quelle einlesen --- *)
axOnline[0] := Anvil.Pfirsich.Status.xOnline;
axOnline[1] := Anvil.Stachelbeere.Status.xOnline;
axOnline[2] := Anvil.Maulbeere.Status.xOnline;
axOnline[3] := Anvil.Felsenbirne.Status.xOnline;
axOnline[4] := Anvil.Maibeere.Status.xOnline;
axOnline[5] := Anvil.Johannisbeere.Status.xOnline;
axOnline[6] := Anvil.Schaltschrank.Status.xOnline;

(* --- 2. Auswerten --- *)
mon(xBmValid := TRUE, axBmOnline := axOnline);

(* --- 3. Nach Bellows durchreichen, damit Hearth es sieht --- *)
Bellows.Diag.auDevState  := mon.auBmState;
Bellows.Diag.asDevStatus := mon.asBmStatus;
Bellows.Diag.xAllOk      := mon.xBmAllOk;
Bellows.Diag.iFaultCount := mon.iBmFaultCount;
Bellows.Diag.sSummary    := mon.sBmSummary;

          
END_PROGRAM

CONFIGURATION config0
  VAR_GLOBAL  (* Pfirsich *)
    xT_2 AT %MX10000.1 : BOOL;  (* Digital input channel 2 (24V DC, opto-isolated) *)
    xT_3 AT %MX10000.2 : BOOL;  (* Digital input channel 3 (24V DC, opto-isolated) *)
  END_VAR
  VAR_GLOBAL  (* Stachelbeere *)
    xT_2 AT %MX10001.1 : BOOL;  (* Digital input channel 2 (24V DC, opto-isolated) *)
    xT_3 AT %MX10001.2 : BOOL;  (* Digital input channel 3 (24V DC, opto-isolated) *)
  END_VAR
  VAR_GLOBAL  (* Maulbeere *)
    xT_2 AT %MX10002.1 : BOOL;  (* Digital input channel 2 (24V DC, opto-isolated) *)
    xT_3 AT %MX10002.2 : BOOL;  (* Digital input channel 3 (24V DC, opto-isolated) *)
  END_VAR
  VAR_GLOBAL  (* Maibeere *)
    xT_2 AT %MX10003.1 : BOOL;  (* Digital input channel 2 (24V DC, opto-isolated) *)
    xT_3 AT %MX10003.2 : BOOL;  (* Digital input channel 3 (24V DC, opto-isolated) *)
  END_VAR
  VAR_GLOBAL  (* Johannisbeere *)
    xT_2 AT %MX10004.1 : BOOL;  (* Digital input channel 2 (24V DC, opto-isolated) *)
    xT_3 AT %MX10004.2 : BOOL;  (* Digital input channel 3 (24V DC, opto-isolated) *)
  END_VAR
  VAR_GLOBAL  (* Felsenbirne *)
    xT_2 AT %MX10005.1 : BOOL;  (* Digital input channel 2 (24V DC, opto-isolated) *)
    xT_3 AT %MX10005.2 : BOOL;  (* Digital input channel 3 (24V DC, opto-isolated) *)
  END_VAR
  VAR_GLOBAL  (* Schrittkette *)
    uRunState AT %MB3 : USINT;  (* Lauf-Zustand der One-Shot-Schrittkette: 0=Idle, 1=Running, 2=Paused, 3=Done. Von PLC_PRG geschrieben, vom HMI nur gelesen. Anwahl allein bewaessert nicht mehr — erst Start armt. *)
  END_VAR
  VAR_GLOBAL  (* Betrieb *)
    aValveJobs AT %MD0 : ARRAY[0..23] OF ST_BedCfg;  (* Job-Liste je Ventil, Index z*4+v (0..23) wie astValveStatus: Pfirsich 0-3, Stachelbeere 4-7, Maulbeere 8-11, Felsenbirne 12-15, Maibeere 16-19, Johannisbeere 20-23. Je Eintrag Anwahl, Startzeit (Stunde/Minute, Ortszeit) und Dauer (ST_BedCfg). Grundlage fuer One-Shot und wiederkehrend. Startzeit und Dauer setzt die HMI, die Anwahl fuehrt FB_SCHEDULE. Die Restzeit steht NICHT hier, sondern im nicht persistenten astValveStatus[i].remainingLiquidation. Persistent: uebersteht Neustart und Programm-Download. *)
    bWeekMask AT %MB1 : BYTE;  (* Wochentag-Freigabe fuer den wiederkehrenden Betrieb (Betriebsart 3): Bit 0 = Montag bis Bit 6 = Sonntag, ein gesetztes Bit gibt den Tag frei. Von der HMI gesetzt, persistent. *)
    astValveStatus AT %MD8 : ARRAY[0..23] OF ST_ValveStatus;  (* Status je Ventil, Index z*4+v: bMode traegt je Betriebsart ein Bit (1 Manuell, 2 One-Shot, 4 wiederkehrend, 8 Auto) — jeder Modus-Baustein setzt sein Bit in einer FOR-Schleife. *)
  END_VAR
  RESOURCE resource0 ON PLC
    TASK task0(INTERVAL := T#20ms, PRIORITY := 0);
    TASK taskDiag(INTERVAL := T#200ms, PRIORITY := 10);
    PROGRAM instance0 WITH task0 : PLC_PRG;
    PROGRAM instBusMonitor WITH taskDiag : BusMonitor;
  END_RESOURCE
END_CONFIGURATION
